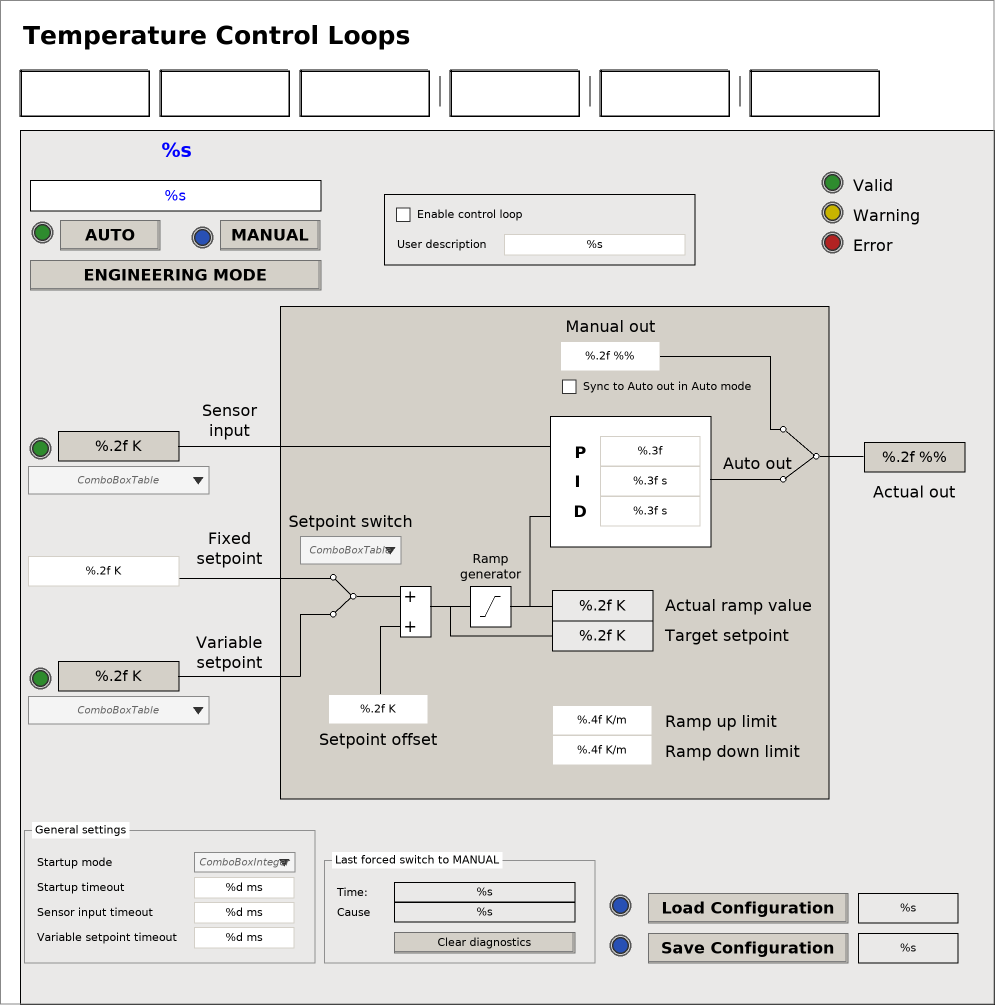
VISUALIZATION VISU_HMI_CRY_TCTRL  // 995x1005
VAR_IN_OUT
	m_Instance : FB_METIS_TCTRL;
    m_Hmi : FB_HMI_CRY_TCTRL;
    m_temp : FB_METIS_TEMPERATURES;
END_VAR
    Rectangle (20,130 975x875)
    Frame (20,70 131x48)
        shows VISU_HMI_SUBSYSTEM_BUTTON(m_Hmi := m_Hmi.tc_cry_sha_button)
        OnMouseClick: execute { m_Hmi.eActiveTab := E_HMI_CRY_TC_TABS.TC_CRY_SHA; }
    Frame (160,70 131x48)
        shows VISU_HMI_SUBSYSTEM_BUTTON(m_Hmi := m_Hmi.tc_cry_shb_button)
        OnMouseClick: execute { m_Hmi.eActiveTab := E_HMI_CRY_TC_TABS.TC_CRY_SHB; }
    Frame (300,70 131x48)
        shows VISU_HMI_SUBSYSTEM_BUTTON(m_Hmi := m_Hmi.tc_cry_shc_button)
        OnMouseClick: execute { m_Hmi.eActiveTab := E_HMI_CRY_TC_TABS.TC_CRY_SHC; }
    Frame (450,70 131x48)
        shows VISU_HMI_SUBSYSTEM_BUTTON(m_Hmi := m_Hmi.tc_cry_pt_button)
        OnMouseClick: execute { m_Hmi.eActiveTab := E_HMI_CRY_TC_TABS.TC_CRY_PT; }
    Line (440,106) (440,76)
    Line (590,106) (590,76)
    Frame (600,70 131x48)
        shows VISU_HMI_SUBSYSTEM_BUTTON(m_Hmi := m_Hmi.tc_cry_wi_button)
        OnMouseClick: execute { m_Hmi.eActiveTab := E_HMI_CRY_TC_TABS.TC_CRY_WI; }
    Frame (20,130 975x875), frame switch variable: m_Hmi.eActiveTab
        shows TEMPLATE_METIS_CTRL_TEMPERATURE(m_instance := m_Instance.tc_cry_sha, m_temp := m_temp)
        shows TEMPLATE_METIS_CTRL_TEMPERATURE(m_instance := m_Instance.tc_cry_shb, m_temp := m_temp)
        shows TEMPLATE_METIS_CTRL_TEMPERATURE(m_instance := m_Instance.tc_cry_shc, m_temp := m_temp)
        shows TEMPLATE_METIS_CTRL_TEMPERATURE(m_instance := m_Instance.tc_cry_pt, m_temp := m_temp)
        shows TEMPLATE_METIS_CTRL_TEMPERATURE(m_instance := m_Instance.tc_cry_wi, m_temp := m_temp)
        shows TEMPLATE_METIS_CTRL_TEMPERATURE(m_instance := m_Instance.tc_cry_sp, m_temp := m_temp)
    Frame (750,70 131x48)
        shows VISU_HMI_SUBSYSTEM_BUTTON(m_Hmi := m_Hmi.tc_cry_sp_button)
        OnMouseClick: execute { m_Hmi.eActiveTab := E_HMI_CRY_TC_TABS.TC_CRY_SP; }
    Line (740,106) (740,76)
    Label (20,20 411x30), "Temperature Control Loops"
END_VISUALIZATION

// HMI/VISUs/Subsystems/CRY/Components/VISU_HMI_CRY_TEMPERATURES
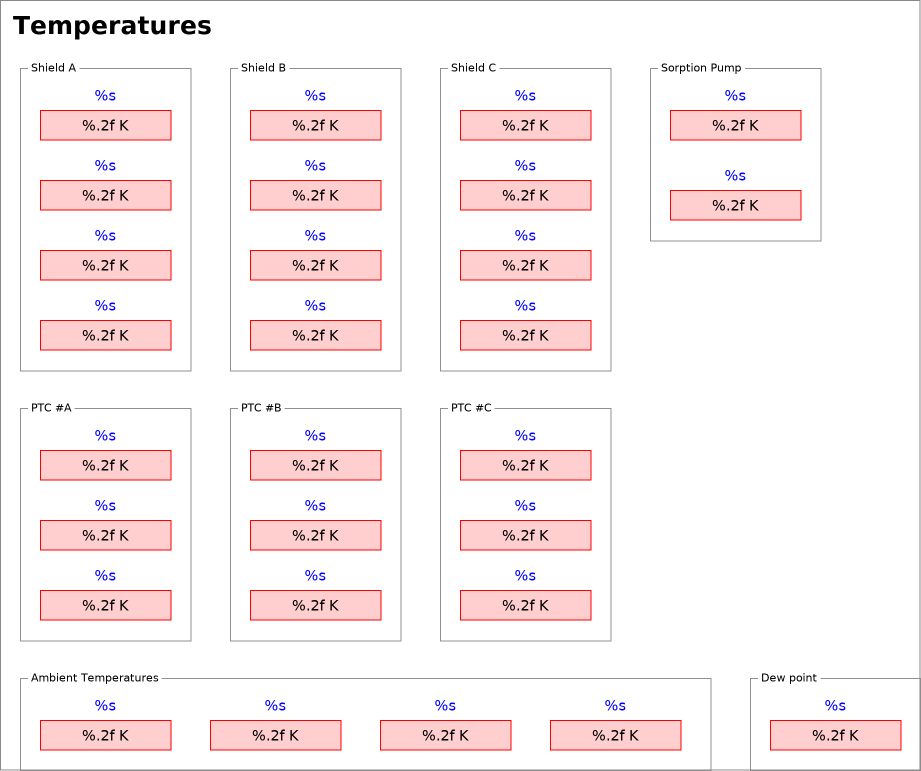
VISUALIZATION VISU_HMI_CRY_TEMPERATURES  // 921x771
VAR_IN_OUT
	m_Instance : FB_METIS_TEMPERATURES;
END_VAR
    Label (10,10 299x30), "Temperatures"
    GroupBox (20,60 171x311), "Shield A"
        Frame (10,20 150x70)
            shows TEMPLATE_TEMP_SENSOR_VALUE_ONLY(m_instance := m_Instance.t_cry_sha_1)
        Frame (10,90 150x70)
            shows TEMPLATE_TEMP_SENSOR_VALUE_ONLY(m_instance := m_Instance.t_cry_sha_2)
        Frame (10,160 150x70)
            shows TEMPLATE_TEMP_SENSOR_VALUE_ONLY(m_instance := m_Instance.t_cry_sha_3)
        Frame (10,230 150x70)
            shows TEMPLATE_TEMP_SENSOR_VALUE_ONLY(m_instance := m_Instance.t_cry_sha_4)
    GroupBox (20,400 171x241), "PTC #A"
        Frame (10,20 150x70)
            shows TEMPLATE_TEMP_SENSOR_VALUE_ONLY(m_instance := m_Instance.t_cry_pta_1)
        Frame (10,90 150x70)
            shows TEMPLATE_TEMP_SENSOR_VALUE_ONLY(m_instance := m_Instance.t_cry_pta_2)
        Frame (10,160 150x70)
            shows TEMPLATE_TEMP_SENSOR_VALUE_ONLY(m_instance := m_Instance.t_cry_pta_3)
    GroupBox (230,60 171x311), "Shield B"
        Frame (10,20 150x70)
            shows TEMPLATE_TEMP_SENSOR_VALUE_ONLY(m_instance := m_Instance.t_cry_shb_1)
        Frame (10,90 150x70)
            shows TEMPLATE_TEMP_SENSOR_VALUE_ONLY(m_instance := m_Instance.t_cry_shb_2)
        Frame (10,160 150x70)
            shows TEMPLATE_TEMP_SENSOR_VALUE_ONLY(m_instance := m_Instance.t_cry_shb_3)
        Frame (10,230 150x70)
            shows TEMPLATE_TEMP_SENSOR_VALUE_ONLY(m_instance := m_Instance.t_cry_shb_4)
    GroupBox (230,400 171x241), "PTC #B"
        Frame (10,20 150x70)
            shows TEMPLATE_TEMP_SENSOR_VALUE_ONLY(m_instance := m_Instance.t_cry_ptb_1)
        Frame (10,90 150x70)
            shows TEMPLATE_TEMP_SENSOR_VALUE_ONLY(m_instance := m_Instance.t_cry_ptb_2)
        Frame (10,160 150x70)
            shows TEMPLATE_TEMP_SENSOR_VALUE_ONLY(m_instance := m_Instance.t_cry_ptb_3)
    GroupBox (440,60 171x311), "Shield C"
        Frame (10,230 150x70)
            shows TEMPLATE_TEMP_SENSOR_VALUE_ONLY(m_instance := m_Instance.t_cry_shc_4)
        Frame (10,160 150x70)
            shows TEMPLATE_TEMP_SENSOR_VALUE_ONLY(m_instance := m_Instance.t_cry_shc_3)
        Frame (10,90 150x70)
            shows TEMPLATE_TEMP_SENSOR_VALUE_ONLY(m_instance := m_Instance.t_cry_shc_2)
        Frame (10,20 150x70)
            shows TEMPLATE_TEMP_SENSOR_VALUE_ONLY(m_instance := m_Instance.t_cry_shc_1)
    GroupBox (440,400 171x241), "PTC #C"
        Frame (10,20 150x70)
            shows TEMPLATE_TEMP_SENSOR_VALUE_ONLY(m_instance := m_Instance.t_cry_ptc_1)
        Frame (10,90 150x70)
            shows TEMPLATE_TEMP_SENSOR_VALUE_ONLY(m_instance := m_Instance.t_cry_ptc_2)
        Frame (10,160 150x70)
            shows TEMPLATE_TEMP_SENSOR_VALUE_ONLY(m_instance := m_Instance.t_cry_ptc_3)
    GroupBox (650,60 171x181), "Sorption Pump"
        Frame (10,20 150x70)
            shows TEMPLATE_TEMP_SENSOR_VALUE_ONLY(m_instance := m_Instance.t_cry_sp_1)
        Frame (10,100 150x70)
            shows TEMPLATE_TEMP_SENSOR_VALUE_ONLY(m_instance := m_Instance.t_cry_sp_2)
    GroupBox (20,670 691x101), "Ambient Temperatures"
        Frame (10,20 150x70)
            shows TEMPLATE_TEMP_SENSOR_VALUE_ONLY(m_instance := m_Instance.t_cry_pca)
        Frame (180,20 150x70)
            shows TEMPLATE_TEMP_SENSOR_VALUE_ONLY(m_instance := m_Instance.t_cry_pcb)
        Frame (350,20 150x70)
            shows TEMPLATE_TEMP_SENSOR_VALUE_ONLY(m_instance := m_Instance.t_cry_wim)
        Frame (520,20 150x70)
            shows TEMPLATE_TEMP_SENSOR_VALUE_ONLY(m_instance := m_Instance.t_cry_wia)
    GroupBox (750,670 171x101), "Dew point"
        Frame (10,20 150x70)
            shows TEMPLATE_TEMP_SENSOR_VALUE_ONLY(m_instance := m_Instance.t_cry_wid)
END_VISUALIZATION

// HMI/VISUs/Subsystems/CRY/Components/VISU_HMI_CRY_VOTERS
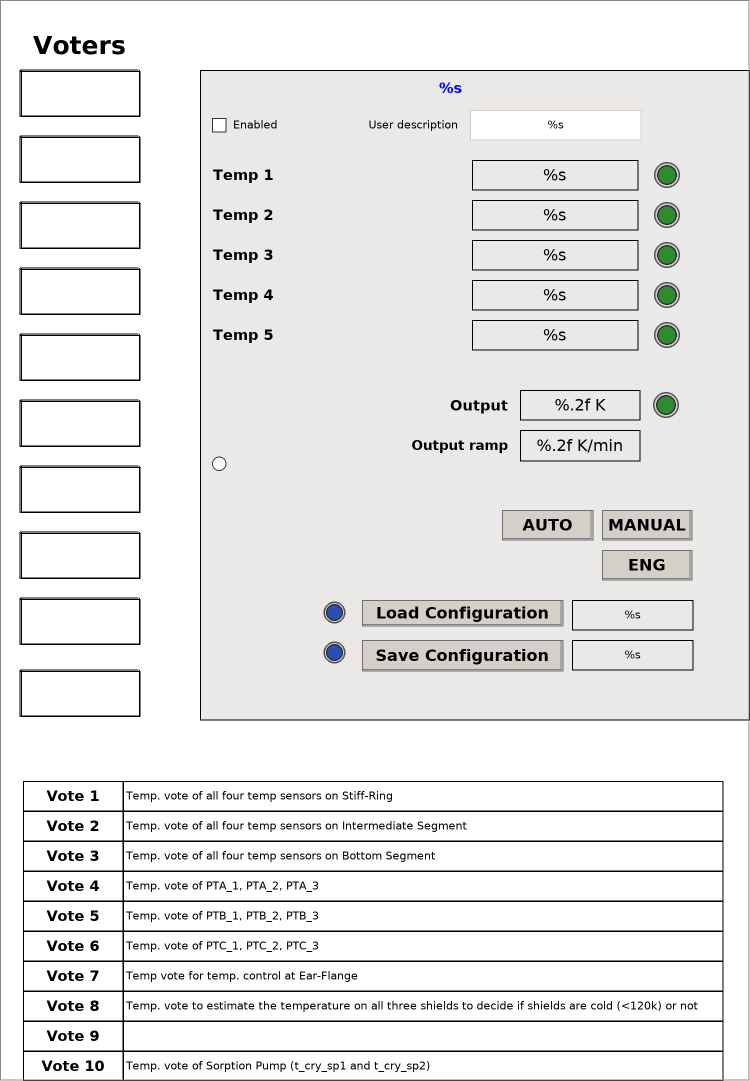
VISUALIZATION VISU_HMI_CRY_VOTERS  // 750x1081
VAR_IN_OUT
    m_Instance : FB_METIS_VOTERS;
	m_Hmi : FB_HMI_CRY_VOTERS;
    m_temperatures : FB_METIS_TEMPERATURES;
END_VAR
    Rectangle (200,70 550x650)
    Frame (20,70 121x48)
        shows VISU_HMI_SUBSYSTEM_BUTTON(m_Hmi := m_Hmi.fbVoter1Button)
        OnMouseClick: execute { m_Hmi.eActiveTab := E_HMI_VOTER_TABS.VOTER_1; }
    Frame (20,136 121x48)
        shows VISU_HMI_SUBSYSTEM_BUTTON(m_Hmi := m_Hmi.fbVoter2Button)
        OnMouseClick: execute { m_Hmi.eActiveTab := E_HMI_VOTER_TABS.VOTER_2; }
    Frame (20,202 121x48)
        shows VISU_HMI_SUBSYSTEM_BUTTON(m_Hmi := m_Hmi.fbVoter3Button)
        OnMouseClick: execute { m_Hmi.eActiveTab := E_HMI_VOTER_TABS.VOTER_3; }
    Frame (20,268 121x48)
        shows VISU_HMI_SUBSYSTEM_BUTTON(m_Hmi := m_Hmi.fbVoter4Button)
        OnMouseClick: execute { m_Hmi.eActiveTab := E_HMI_VOTER_TABS.VOTER_4; }
    Frame (20,334 121x48)
        shows VISU_HMI_SUBSYSTEM_BUTTON(m_Hmi := m_Hmi.fbVoter5Button)
        OnMouseClick: execute { m_Hmi.eActiveTab := E_HMI_VOTER_TABS.VOTER_5; }
    Frame (20,400 121x48)
        shows VISU_HMI_SUBSYSTEM_BUTTON(m_Hmi := m_Hmi.fbVoter6Button)
        OnMouseClick: execute { m_Hmi.eActiveTab := E_HMI_VOTER_TABS.VOTER_6; }
    Frame (20,466 121x48)
        shows VISU_HMI_SUBSYSTEM_BUTTON(m_Hmi := m_Hmi.fbVoter7Button)
        OnMouseClick: execute { m_Hmi.eActiveTab := E_HMI_VOTER_TABS.VOTER_7; }
    Frame (20,532 121x48)
        shows VISU_HMI_SUBSYSTEM_BUTTON(m_Hmi := m_Hmi.fbVoter8Button)
        OnMouseClick: execute { m_Hmi.eActiveTab := E_HMI_VOTER_TABS.VOTER_8; }
    Frame (20,598 121x48)
        shows VISU_HMI_SUBSYSTEM_BUTTON(m_Hmi := m_Hmi.fbVoter9Button)
        OnMouseClick: execute { m_Hmi.eActiveTab := E_HMI_VOTER_TABS.VOTER_9; }
    Frame (20,670 121x48)
        shows VISU_HMI_SUBSYSTEM_BUTTON(m_Hmi := m_Hmi.fbVoter10Button)
        OnMouseClick: execute { m_Hmi.eActiveTab := E_HMI_VOTER_TABS.VOTER_10; }
    Frame (200,70 545x641), frame switch variable: m_Hmi.eActiveTab
        shows TEMPLATE_TEMPERATURE_VOTE(m_Instance := m_Instance.vote_cry_1, m_all_temperatures_array := m_temperatures)
        shows TEMPLATE_TEMPERATURE_VOTE(m_Instance := m_Instance.vote_cry_2, m_all_temperatures_array := m_temperatures)
        shows TEMPLATE_TEMPERATURE_VOTE(m_Instance := m_Instance.vote_cry_3, m_all_temperatures_array := m_temperatures)
        shows TEMPLATE_TEMPERATURE_VOTE(m_Instance := m_Instance.vote_cry_4, m_all_temperatures_array := m_temperatures)
        shows TEMPLATE_TEMPERATURE_VOTE(m_Instance := m_Instance.vote_cry_5, m_all_temperatures_array := m_temperatures)
        shows TEMPLATE_TEMPERATURE_VOTE(m_Instance := m_Instance.vote_cry_6, m_all_temperatures_array := m_temperatures)
        shows TEMPLATE_TEMPERATURE_VOTE(m_Instance := m_Instance.vote_cry_7, m_all_temperatures_array := m_temperatures)
        shows TEMPLATE_TEMPERATURE_VOTE(m_Instance := m_Instance.vote_cry_8, m_all_temperatures_array := m_temperatures)
        shows TEMPLATE_TEMPERATURE_VOTE(m_Instance := m_Instance.vote_cry_9, m_all_temperatures_array := m_temperatures)
        shows TEMPLATE_TEMPERATURE_VOTE(m_Instance := m_Instance.vote_cry_10, m_all_temperatures_array := m_temperatures)
    Label (30,30 411x30), "Voters"
    Rectangle (23,781 100x30), "Vote 1"
    Rectangle (123,781 600x30), "Temp. vote of all four temp sensors on Stiff-Ring"
    Rectangle (23,811 100x30), "Vote 2"
    Rectangle (123,811 600x30), "Temp. vote of all four temp sensors on Intermediate Segment"
    Rectangle (23,841 100x30), "Vote 3"
    Rectangle (123,841 600x30), "Temp. vote of all four temp sensors on Bottom Segment"
    Rectangle (23,871 100x30), "Vote 4"
    Rectangle (123,871 600x30), "Temp. vote of PTA_1, PTA_2, PTA_3"
    Rectangle (23,901 100x30), "Vote 5"
    Rectangle (123,901 600x30), "Temp. vote of PTB_1, PTB_2, PTB_3"
    Rectangle (23,931 100x30), "Vote 6"
    Rectangle (123,931 600x30), "Temp. vote of PTC_1, PTC_2, PTC_3"
    Rectangle (23,961 100x30), "Vote 7"
    Rectangle (123,961 600x30), "Temp vote for temp. control at Ear-Flange"
    Rectangle (23,991 100x30), "Vote 8"
    Rectangle (123,991 600x30), "Temp. vote to estimate the temperature on all three shields to decide if shields are cold (<120k) or not"
    Rectangle (23,1021 100x30), "Vote 9"
    Rectangle (123,1021 600x30)
    Rectangle (23,1051 100x30), "Vote 10"
    Rectangle (123,1051 600x30), "Temp. vote of Sorption Pump (t_cry_sp1 and t_cry_sp2)"
END_VISUALIZATION

// HMI/VISUs/Subsystems/CRY/VISU_HMI_CRY
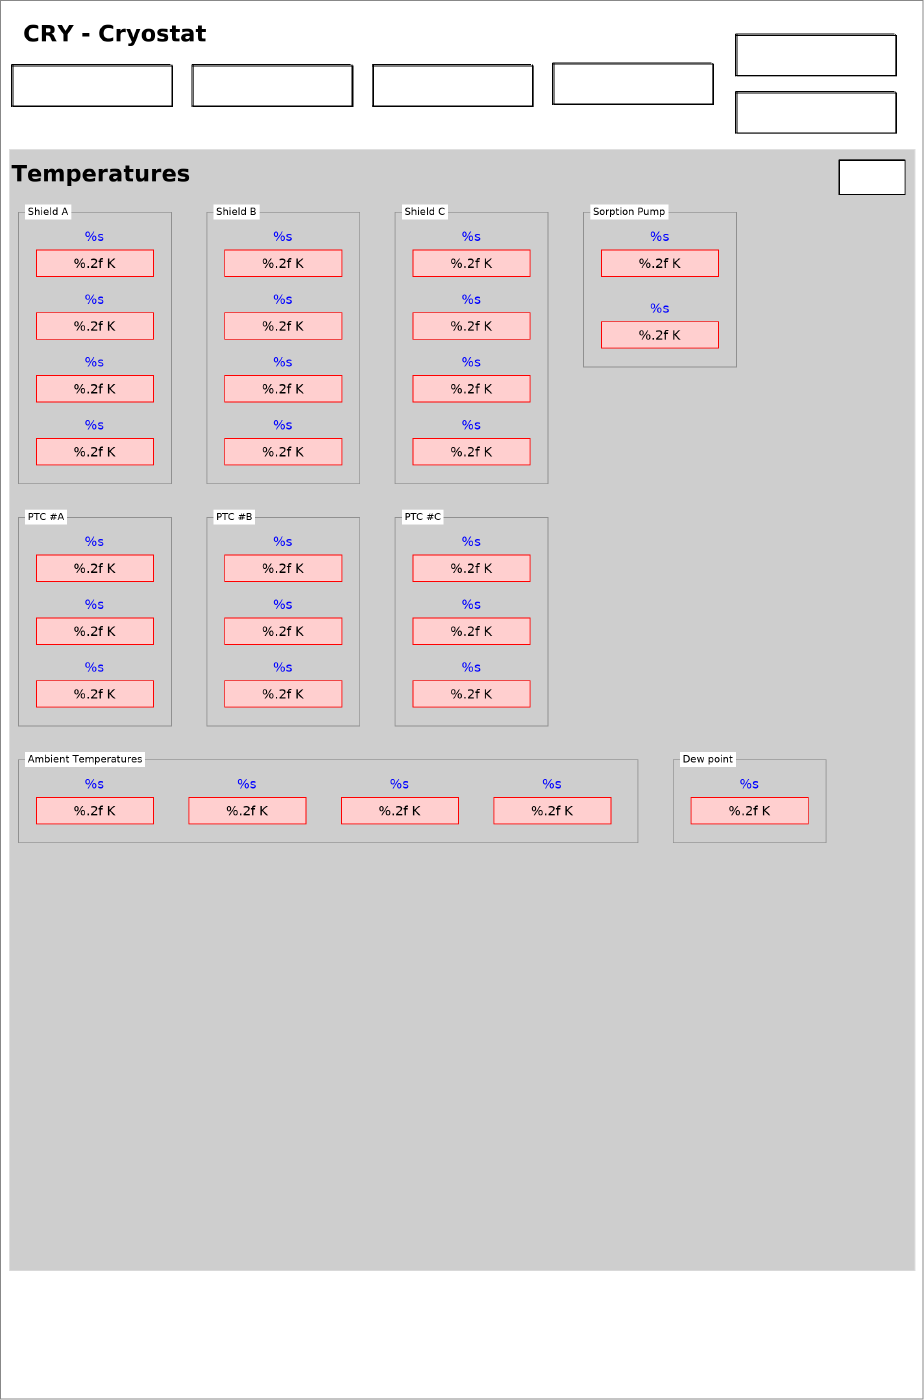
VISUALIZATION VISU_HMI_CRY  // 1030x1560
VAR_IN_OUT
	met_cryo_ctrl: FB_METIS_CRYO_CTRL;
    m_Hmi : FB_HMI_CRY;
END_VAR
    Frame (0,36 1021x1397)
        shows TEMPLATE_BACKGROUND_LEVEL_2()
    Label (23,22 671x30), "CRY - Cryostat"
    Frame (0,168 1017x1250), frame switch variable: m_Hmi.eActiveTab
        shows VISU_HMI_CRY_TEMPERATURES(m_Instance := met_cryo_ctrl.met_temp)
        shows VISU_HMI_CRY_RH(m_Instance := met_cryo_ctrl.met_rh)
        shows VISU_HMI_CRY_HEATERS(m_Instance := met_cryo_ctrl.met_heaters, m_Hmi := m_Hmi.fbHeaters)
        shows VISU_HMI_CRY_VOTERS(m_Instance := met_cryo_ctrl.met_voters, m_Hmi := m_Hmi.fbVoters, m_temperatures := met_cryo_ctrl.met_temp)
        shows VISU_HMI_CRY_TCTRL(m_Instance := met_cryo_ctrl.met_tctrl, m_Hmi := m_Hmi.fbTControl, m_temp := met_cryo_ctrl.met_temp)
        shows VISU_HMI_CRY_LN2_LEVEL_CONTROL()
    Frame (13,72 181x48)
        shows VISU_HMI_SUBSYSTEM_BUTTON(m_Hmi := m_Hmi.fbTemperaturesButton)
        OnMouseClick: execute { m_Hmi.eActiveTab := E_HMI_CRY_TABS.TEMPERATURES; }
    Frame (616,70 181x48)
        shows VISU_HMI_SUBSYSTEM_BUTTON(m_Hmi := m_Hmi.fbHeatersButton)
        OnMouseClick: execute { m_Hmi.eActiveTab := E_HMI_CRY_TABS.HEATERS; }
    Frame (214,72 181x48)
        shows VISU_HMI_SUBSYSTEM_BUTTON(m_Hmi := m_Hmi.fbVotersButton)
        OnMouseClick: execute { m_Hmi.eActiveTab := E_HMI_CRY_TABS.VOTERS; }
    Frame (415,72 181x48)
        shows VISU_HMI_SUBSYSTEM_BUTTON(m_Hmi := m_Hmi.fbTControlButton)
        OnMouseClick: execute { m_Hmi.eActiveTab := E_HMI_CRY_TABS.TCONTROL; }
    Group (820,38 181x112)
        Frame (0,0 181x48)
            shows VISU_HMI_SUBSYSTEM_BUTTON(m_Hmi := m_Hmi.fbRhButton)
            OnMouseClick: execute { m_Hmi.eActiveTab := E_HMI_CRY_TABS.RH; }
        Frame (0,64 181x48)
            shows VISU_HMI_SUBSYSTEM_BUTTON(m_Hmi := m_Hmi.fbLN2ControlButton)
            OnMouseClick: execute { m_Hmi.eActiveTab := E_HMI_CRY_TABS.LN2CONTROL; }
    Frame (935,178 75x40)
        shows VISU_HMI_SUBSYSTEM_BUTTON(m_Hmi := PRG_HMI.fbBackButton)
        OnMouseClick: execute { PRG_HMI.eActiveTab := PRG_HMI.ePreviousTab; }
END_VISUALIZATION

// HMI/VISUs/Subsystems/ICS/Components/VISU_HMI_ICS_CCU_CONFIGS
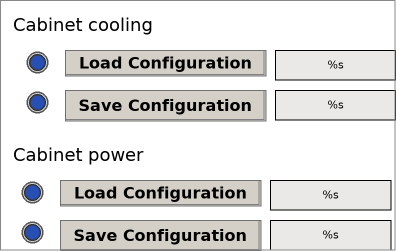
VISUALIZATION VISU_HMI_ICS_CCU_CONFIGS  // 396x251
VAR_IN_OUT
	m_CoolingCfg : FB_READ_WRITE_CAB_COOLING_CONFIG;
    m_PowerCfg : FB_READ_WRITE_CAB_POWER_CONFIG;
END_VAR
    Lamp1 (25,50 25x25), tooltip "Command coming from the Control System", variable: m_CoolingCfg.bReading, style: Lamp-Lamp1-Blue
    Button (65,90 201x31), "Save Configuration"
        OnMouseClick: execute { m_CoolingCfg.M_WriteConfiguration(); }
    Button (65,50 201x26), "Load Configuration"
        OnMouseClick: execute { m_CoolingCfg.M_ReadConfiguration(); }
    Lamp1 (25,90 25x25), tooltip "Command coming from the Control System", variable: m_CoolingCfg.bWriting, style: Lamp-Lamp1-Blue
    Rectangle (275,50 121x30), "%s", text variable: m_CoolingCfg.sReadError, colour toggle: m_CoolingCfg.bReadError
    Rectangle (275,90 121x30), "%s", text variable: m_CoolingCfg.sWriteError, colour toggle: m_CoolingCfg.bWriteError
    Label (10,10 206x30), "Cabinet cooling"
    Label (10,140 206x30), "Cabinet power"
    Lamp1 (20,180 25x25), variable: m_PowerCfg.bReading, style: Lamp-Lamp1-Blue
    Button (60,220 201x31), "Save Configuration"
        OnMouseClick: execute { m_PowerCfg.M_WriteConfiguration(); }
    Button (60,180 201x26), "Load Configuration"
        OnMouseClick: execute { m_PowerCfg.M_ReadConfiguration(); }
    Lamp1 (20,220 25x25), tooltip "Command coming from the Control System", variable: m_PowerCfg.bWriting, style: Lamp-Lamp1-Blue
    Rectangle (270,180 121x30), "%s", text variable: m_PowerCfg.sReadError, colour toggle: m_PowerCfg.bReadError
    Rectangle (270,220 121x30), "%s", text variable: m_PowerCfg.sWriteError, colour toggle: m_PowerCfg.bWriteError
END_VISUALIZATION

// HMI/VISUs/Subsystems/ICS/Components/VISU_HMI_ICS_CCUS_CONFIGS
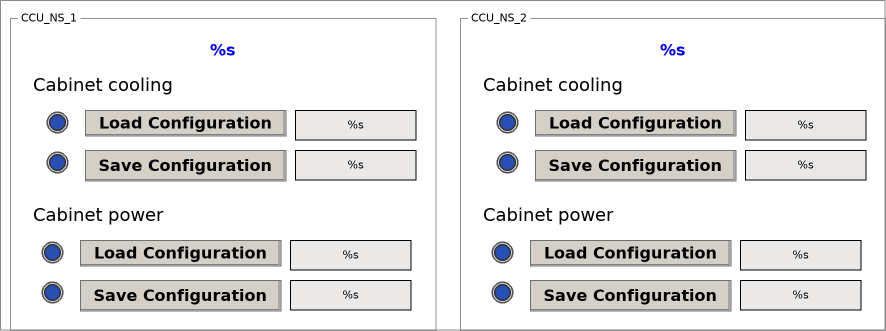
VISUALIZATION VISU_HMI_ICS_CCUS_CONFIGS  // 886x331
VAR_IN_OUT
	m_CCUs : FB_METIS_CCUS;
    m_Hmi : FB_HMI_ICS;
END_VAR
    GroupBox (10,10 426x321), "CCU_NS_1"
        Frame (10,50 397x252)
            shows VISU_HMI_ICS_CCU_CONFIGS(m_CoolingCfg := m_CCUs.aCoolingConfig[1], m_PowerCfg := m_CCUs.aPowerConfig[1])
        Rectangle (20,25 386x30), "%s", text variable: m_CCUs.ccu_ns_1.in_sCabinetName
    GroupBox (460,10 426x321), "CCU_NS_2"
        Frame (10,50 397x252)
            shows VISU_HMI_ICS_CCU_CONFIGS(m_CoolingCfg := m_CCUs.aCoolingConfig[2], m_PowerCfg := m_CCUs.aPowerConfig[2])
        Rectangle (20,25 386x30), "%s", text variable: m_CCUs.ccu_ns_2.in_sCabinetName
END_VISUALIZATION

// HMI/VISUs/Subsystems/ICS/VISU_HMI_ICS
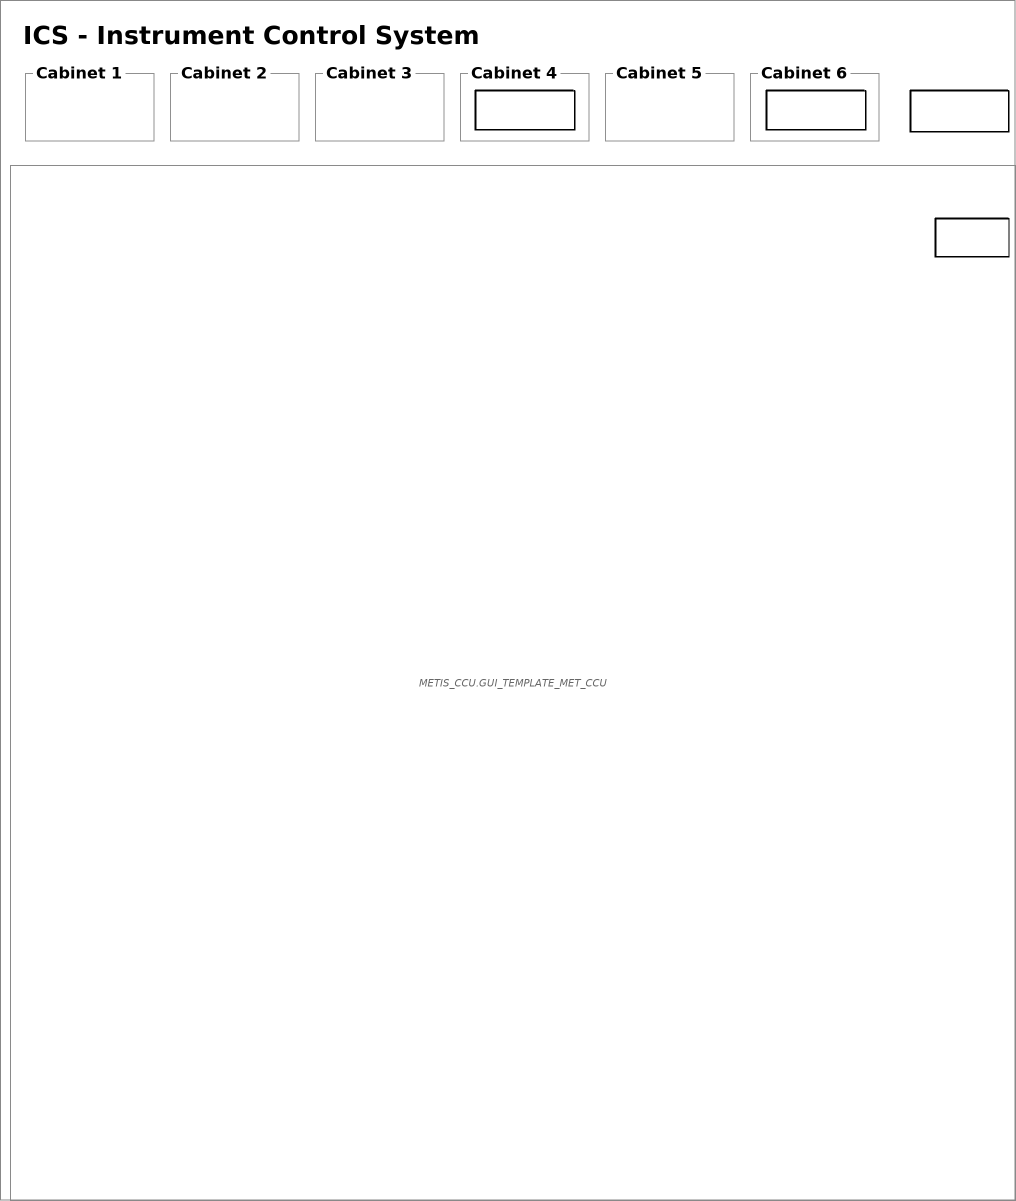
VISUALIZATION VISU_HMI_ICS  // 1016x1201
VAR_IN_OUT
	m_CCUs : FB_METIS_CCUS;
    m_Hmi : FB_HMI_ICS;
END_VAR
    Label (20,20 671x30), "ICS - Instrument Control System"
    Frame (10,165 1006x1036), frame switch variable: m_Hmi.eActiveTab
        shows METIS_CCU.GUI_TEMPLATE_MET_CCU(m_Instance := m_CCUs.ccu_ns_1)
        shows METIS_CCU.GUI_TEMPLATE_MET_CCU(m_Instance := m_CCUs.ccu_ns_2)
        shows VISU_HMI_ICS_CCUS_CONFIGS(m_CCUs := m_CCUs, m_Hmi := m_Hmi)
        shows METIS_CCU.GUI_TEMPLATE_MET_CCU(m_Instance := m_CCUs.ccu_ns_4)
        shows METIS_CCU.GUI_TEMPLATE_MET_CCU(m_Instance := m_CCUs.ccu_ns_5)
        shows METIS_CCU.GUI_TEMPLATE_MET_CCU(m_Instance := m_CCUs.ccu_6)
        shows VISU_HMI_ICS_CCUS_CONFIGS(m_CCUs := m_CCUs, m_Hmi := m_Hmi)
        p4089929901: m_CCUs.ccu_ns_3
    Frame (910,90 100x43)
        shows VISU_HMI_SUBSYSTEM_BUTTON(m_Hmi := m_Hmi.fbConfigsButton)
        shows METIS_CCU.GUI_TEMPLATE_MET_CCU()
        shows METIS_CCU.GUI_TEMPLATE_MET_CCU()
        shows METIS_CCU.GUI_TEMPLATE_MET_CCU()
        shows METIS_CCU.GUI_TEMPLATE_MET_CCU()
        shows METIS_CCU.GUI_TEMPLATE_MET_CCU()
        OnMouseClick: execute { m_Hmi.eActiveTab := E_HMI_ICS_TABS.CCU_CONFIGS; }
    Frame (935,218 75x40)
        shows VISU_HMI_SUBSYSTEM_BUTTON(m_Hmi := PRG_HMI.fbBackButton)
        OnMouseClick: execute { PRG_HMI.eActiveTab := PRG_HMI.ePreviousTab; }
    GroupBox (25,65 129x76), "Cabinet 1"
    GroupBox (170,65 129x76), "Cabinet 2"
    GroupBox (315,65 129x76), "Cabinet 3"
    GroupBox (460,65 129x76), "Cabinet 4"
        Frame (15,25 101x41)
            shows VISU_HMI_SUBSYSTEM_BUTTON(m_Hmi := m_Hmi.fbCCU_NS_2_Button)
            shows METIS_CCU.GUI_TEMPLATE_MET_CCU()
            shows METIS_CCU.GUI_TEMPLATE_MET_CCU()
            shows METIS_CCU.GUI_TEMPLATE_MET_CCU()
            shows METIS_CCU.GUI_TEMPLATE_MET_CCU()
            shows METIS_CCU.GUI_TEMPLATE_MET_CCU()
            OnMouseClick: execute { m_Hmi.eActiveTab := E_HMI_ICS_TABS.CCU_NS_2; }
    GroupBox (605,65 129x76), "Cabinet 5"
    GroupBox (750,65 129x76), "Cabinet 6"
        Frame (16,25 101x41)
            shows VISU_HMI_SUBSYSTEM_BUTTON(m_Hmi := m_Hmi.fbCCU_NS_1_Button)
            shows METIS_CCU.GUI_TEMPLATE_MET_CCU()
            shows METIS_CCU.GUI_TEMPLATE_MET_CCU()
            shows METIS_CCU.GUI_TEMPLATE_MET_CCU()
            shows METIS_CCU.GUI_TEMPLATE_MET_CCU()
            shows METIS_CCU.GUI_TEMPLATE_MET_CCU()
            OnMouseClick: execute { m_Hmi.eActiveTab := E_HMI_ICS_TABS.CCU_NS_1; }
END_VISUALIZATION

// HMI/VISUs/Subsystems/IMG/Components/VISU_HMI_IMG_HEATERS
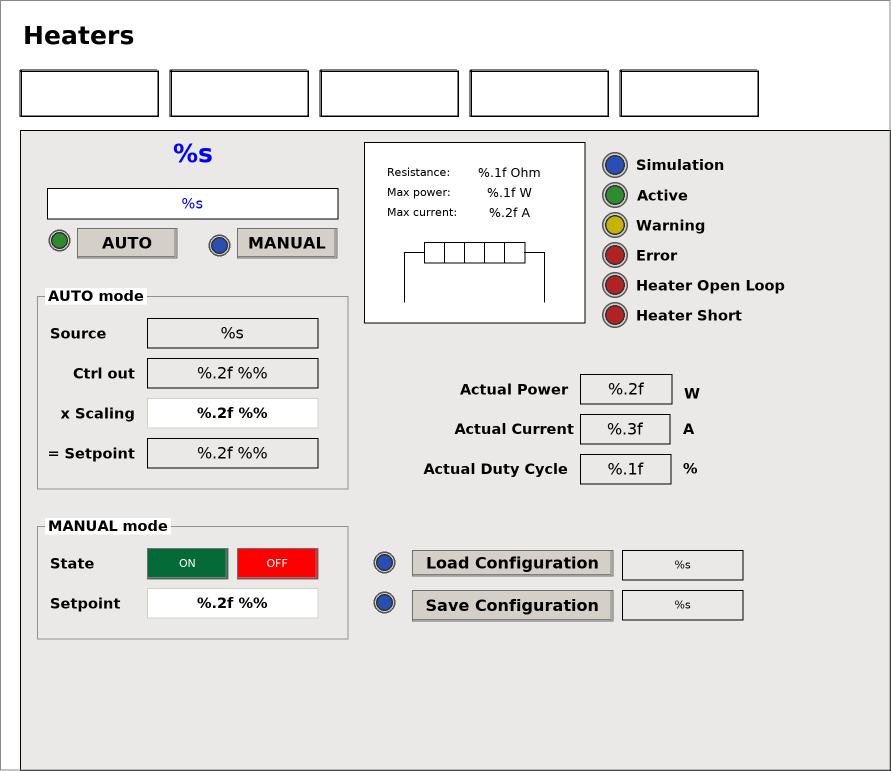
VISUALIZATION VISU_HMI_IMG_HEATERS  // 891x771
VAR_IN_OUT
	m_Instance  : FB_METIS_HEATERS;
    m_Hmi       : FB_HMI_IMG_HEATERS;
END_VAR
    Rectangle (20,130 871x641)
    Label (20,20 411x30), "Heaters"
    Frame (20,130 800x550), frame switch variable: m_Hmi.eActiveTab
        shows TEMPLATE_METIS_HEATER(m_instance := m_Instance.h_img_wuh_1)
        shows TEMPLATE_METIS_HEATER(m_instance := m_Instance.h_img_wuh_2)
        shows TEMPLATE_METIS_HEATER(m_instance := m_Instance.h_img_lmd_2)
        shows TEMPLATE_METIS_HEATER(m_instance := m_Instance.h_img_lmp_2)
        shows TEMPLATE_METIS_HEATER(m_instance := m_Instance.h_img_nd_2)
        shows METIS_Cryo_PLC.TEMPLATE_METIS_CTRL_DT670(m_temp := m_temp)
        p8630679: tcontrol.tc_img_wuh_1
        p371692913: tcontrol.vote_img_wuh_1
        p2286783886: temperatures
    Frame (20,70 140x48)
        shows VISU_HMI_SUBSYSTEM_BUTTON(m_Hmi := m_Hmi.h_img_wuh_1_button)
        OnMouseClick: execute { m_Hmi.eActiveTab := E_HMI_IMG_HEATER_TABS.H_IMG_WUH_1; }
    Frame (170,70 140x48)
        shows VISU_HMI_SUBSYSTEM_BUTTON(m_Hmi := m_Hmi.h_img_wuh_2_button)
        OnMouseClick: execute { m_Hmi.eActiveTab := E_HMI_IMG_HEATER_TABS.H_IMG_WUH_2; }
    Frame (320,70 140x48)
        shows VISU_HMI_SUBSYSTEM_BUTTON(m_Hmi := m_Hmi.h_img_lmd_2_button)
        OnMouseClick: execute { m_Hmi.eActiveTab := E_HMI_IMG_HEATER_TABS.H_IMG_LMD_2; }
    Frame (470,70 140x48)
        shows VISU_HMI_SUBSYSTEM_BUTTON(m_Hmi := m_Hmi.h_img_lmp_2_button)
        OnMouseClick: execute { m_Hmi.eActiveTab := E_HMI_IMG_HEATER_TABS.H_IMG_LMP_2; }
    Frame (620,70 140x48)
        shows VISU_HMI_SUBSYSTEM_BUTTON(m_Hmi := m_Hmi.h_img_nd_2_button)
        OnMouseClick: execute { m_Hmi.eActiveTab := E_HMI_IMG_HEATER_TABS.H_IMG_ND_2; }
END_VISUALIZATION

// HMI/VISUs/Subsystems/IMG/Components/VISU_HMI_IMG_TC
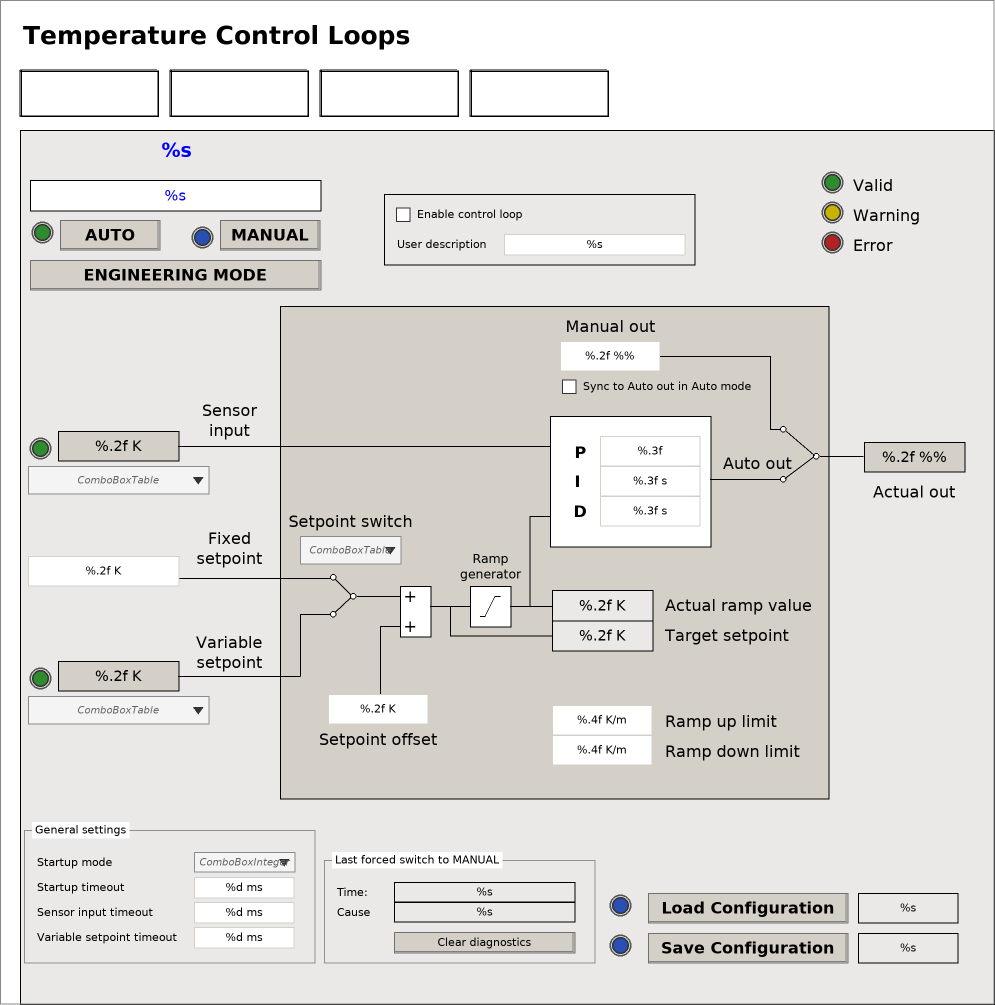
VISUALIZATION VISU_HMI_IMG_TC  // 995x1005
VAR_IN_OUT
    m_Instance : FB_METIS_TCTRL;
    m_Hmi : FB_HMI_IMG_TCTRL;
    m_temp : FB_METIS_TEMPERATURES;
END_VAR
    Rectangle (20,130 975x875)
    Label (20,20 411x30), "Temperature Control Loops"
    Frame (20,130 975x875), frame switch variable: m_Hmi.eActiveTab
        shows TEMPLATE_METIS_CTRL_TEMPERATURE(m_instance := m_Instance.tc_img_wuh, m_temp := m_temp)
        shows TEMPLATE_METIS_CTRL_TEMPERATURE(m_instance := m_Instance.tc_img_lmd_2, m_temp := m_temp)
        shows TEMPLATE_METIS_CTRL_TEMPERATURE(m_instance := m_Instance.tc_img_lmp_2, m_temp := m_temp)
        shows TEMPLATE_METIS_CTRL_TEMPERATURE(m_instance := m_Instance.tc_img_nd_2, m_temp := m_temp)
        shows METIS_Cryo_PLC.TEMPLATE_METIS_CTRL_DT670(m_temp := m_temp)
        p8630679: tcontrol.tc_img_wuh_1
        p371692913: tcontrol.vote_img_wuh_1
        p2286783886: temperatures
        p2857688358: m_Instance.tc_img_nd_2
        p3792852128: m_temp
    Frame (20,70 140x48)
        shows VISU_HMI_SUBSYSTEM_BUTTON(m_Hmi := m_Hmi.tc_img_wuh_button)
        OnMouseClick: execute { m_Hmi.eActiveTab := E_HMI_IMG_TC_TABS.TC_IMG_WUH; }
    Frame (170,70 140x48)
        shows VISU_HMI_SUBSYSTEM_BUTTON(m_Hmi := m_Hmi.tc_img_lmd_2_button)
        OnMouseClick: execute { m_Hmi.eActiveTab := E_HMI_IMG_TC_TABS.TC_IMG_LMD_2; }
    Frame (320,70 140x48)
        shows VISU_HMI_SUBSYSTEM_BUTTON(m_Hmi := m_Hmi.tc_img_lmp_2_button)
        OnMouseClick: execute { m_Hmi.eActiveTab := E_HMI_IMG_TC_TABS.TC_IMG_LMP_2; }
    Frame (470,70 140x48)
        shows VISU_HMI_SUBSYSTEM_BUTTON(m_Hmi := m_Hmi.tc_img_nd_2_button)
        OnMouseClick: execute { m_Hmi.eActiveTab := E_HMI_IMG_TC_TABS.TC_IMG_ND_2; }
END_VISUALIZATION

// HMI/VISUs/Subsystems/IMG/Components/VISU_HMI_IMG_TEMPERATURES
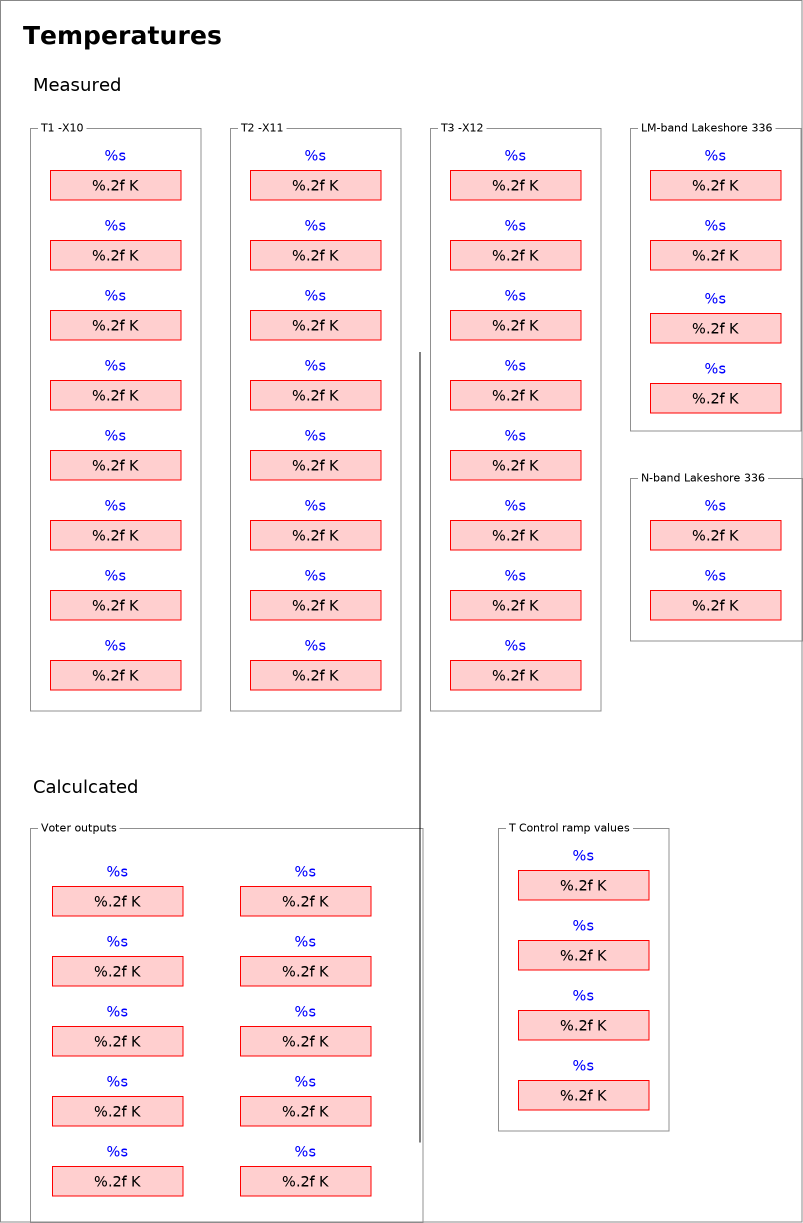
VISUALIZATION VISU_HMI_IMG_TEMPERATURES  // 803x1223
VAR_IN_OUT
	m_Instance : FB_METIS_TEMPERATURES;
END_VAR
    GroupBox (230,120 171x591), "T2 -X11"
        Frame (10,20 150x70)
            shows TEMPLATE_TEMP_SENSOR_VALUE_ONLY(m_instance := m_Instance.t_img_npw_1)
        Frame (10,90 150x70)
            shows TEMPLATE_TEMP_SENSOR_VALUE_ONLY(m_instance := m_Instance.t_img_npw_2)
        Frame (10,160 150x70)
            shows TEMPLATE_TEMP_SENSOR_VALUE_ONLY(m_instance := m_Instance.t_img_nfw_1)
        Frame (10,230 150x70)
            shows TEMPLATE_TEMP_SENSOR_VALUE_ONLY(m_instance := m_Instance.t_img_nfw_2)
        Frame (10,300 150x70)
            shows TEMPLATE_TEMP_SENSOR_VALUE_ONLY(m_instance := m_Instance.t_img_npr_1)
        Frame (10,370 150x70)
            shows TEMPLATE_TEMP_SENSOR_VALUE_ONLY(m_instance := m_Instance.t_img_bwu_2)
        Frame (10,440 150x70)
            shows TEMPLATE_TEMP_SENSOR_VALUE_ONLY(m_instance := m_Instance.t_img_nnd_1)
        Frame (10,510 150x70)
            shows TEMPLATE_TEMP_SENSOR_VALUE_ONLY(m_instance := m_Instance.t_img_nnd_2)
    GroupBox (30,120 171x591), "T1 -X10"
        Frame (10,20 150x70)
            shows TEMPLATE_TEMP_SENSOR_VALUE_ONLY(m_instance := m_Instance.t_img_lpw_1)
        Frame (10,90 150x70)
            shows TEMPLATE_TEMP_SENSOR_VALUE_ONLY(m_instance := m_Instance.t_img_lpw_2)
        Frame (10,160 150x70)
            shows TEMPLATE_TEMP_SENSOR_VALUE_ONLY(m_instance := m_Instance.t_img_lfw_1)
        Frame (10,230 150x70)
            shows TEMPLATE_TEMP_SENSOR_VALUE_ONLY(m_instance := m_Instance.t_img_lfw_2)
        Frame (10,300 150x70)
            shows TEMPLATE_TEMP_SENSOR_VALUE_ONLY(m_instance := m_Instance.t_img_lpr_1)
        Frame (10,370 150x70)
            shows TEMPLATE_TEMP_SENSOR_VALUE_ONLY(m_instance := m_Instance.t_img_bwu_3)
        Frame (10,440 150x70)
            shows TEMPLATE_TEMP_SENSOR_VALUE_ONLY(m_instance := m_Instance.t_img_lnd_1)
        Frame (10,510 150x70)
            shows TEMPLATE_TEMP_SENSOR_VALUE_ONLY(m_instance := m_Instance.t_img_lnd_2)
    Label (20,20 299x30), "Temperatures"
    GroupBox (430,120 171x591), "T3 -X12"
        Frame (10,20 150x70)
            shows TEMPLATE_TEMP_SENSOR_VALUE_ONLY(m_instance := m_Instance.t_img_opt_1)
        Frame (10,90 150x70)
            shows TEMPLATE_TEMP_SENSOR_VALUE_ONLY(m_instance := m_Instance.t_img_bwu_1)
        Frame (10,160 150x70)
            shows TEMPLATE_TEMP_SENSOR_VALUE_ONLY(m_instance := m_Instance.t_img_ctr_1)
        Frame (10,230 150x70)
            shows TEMPLATE_TEMP_SENSOR_VALUE_ONLY(m_instance := m_Instance.t_img_ctr_2)
        Frame (10,300 150x70)
            shows TEMPLATE_TEMP_SENSOR_VALUE_ONLY(m_instance := m_Instance.t_img_70k_1)
        Frame (10,370 150x70)
            shows TEMPLATE_TEMP_SENSOR_VALUE_ONLY(m_instance := m_Instance.t_img_ln2_1)
        Frame (10,440 150x70)
            shows TEMPLATE_TEMP_SENSOR_VALUE_ONLY(m_instance := m_Instance.t_img_ln2_2)
        Frame (10,510 150x70)
            shows TEMPLATE_TEMP_SENSOR_VALUE_ONLY(m_instance := m_Instance.t_img_hex_1)
    GroupBox (630,120 171x311), "LM-band Lakeshore 336"
        Frame (10,20 150x70)
            shows TEMPLATE_TEMP_SENSOR_VALUE_ONLY(m_instance := m_Instance.t_img_lmd_1)
        Frame (10,90 150x70)
            shows TEMPLATE_TEMP_SENSOR_VALUE_ONLY(m_instance := m_Instance.t_img_lmd_2)
        Frame (10,163 150x70)
            shows TEMPLATE_TEMP_SENSOR_VALUE_ONLY(m_instance := m_Instance.t_img_lmp_1)
        Frame (10,233 150x70)
            shows TEMPLATE_TEMP_SENSOR_VALUE_ONLY(m_instance := m_Instance.t_img_lmp_2)
    GroupBox (630,470 173x171), "N-band Lakeshore 336"
        Frame (10,20 150x70)
            shows TEMPLATE_TEMP_SENSOR_VALUE_ONLY(m_instance := m_Instance.t_img_nd_1)
        Frame (10,90 150x70)
            shows TEMPLATE_TEMP_SENSOR_VALUE_ONLY(m_instance := m_Instance.t_img_nd_2)
    GroupBox (30,820 393x403), "Voter outputs"
        Group (12,36 150x350)
            Frame (0,0 150x70)
                shows TEMPLATE_TEMP_SENSOR_VALUE_ONLY(m_instance := m_Instance.t_img_vot_1)
            Frame (0,70 150x70)
                shows TEMPLATE_TEMP_SENSOR_VALUE_ONLY(m_instance := m_Instance.t_img_vot_2)
            Frame (0,140 150x70)
                shows TEMPLATE_TEMP_SENSOR_VALUE_ONLY(m_instance := m_Instance.t_img_vot_3)
            Frame (0,210 150x70)
                shows TEMPLATE_TEMP_SENSOR_VALUE_ONLY(m_instance := m_Instance.t_img_vot_4)
            Frame (0,280 150x70)
                shows TEMPLATE_TEMP_SENSOR_VALUE_ONLY(m_instance := m_Instance.t_img_vot_5)
        Group (200,36 150x350)
            Frame (0,0 150x70)
                shows TEMPLATE_TEMP_SENSOR_VALUE_ONLY(m_instance := m_Instance.t_img_vot_6)
            Frame (0,70 150x70)
                shows TEMPLATE_TEMP_SENSOR_VALUE_ONLY(m_instance := m_Instance.t_img_vot_7)
            Frame (0,140 150x70)
                shows TEMPLATE_TEMP_SENSOR_VALUE_ONLY(m_instance := m_Instance.t_img_vot_8)
            Frame (0,210 150x70)
                shows TEMPLATE_TEMP_SENSOR_VALUE_ONLY(m_instance := m_Instance.t_img_vot_9)
            Frame (0,280 150x70)
                shows TEMPLATE_TEMP_SENSOR_VALUE_ONLY(m_instance := m_Instance.t_img_vot_10)
    GroupBox (498,820 171x311), "T Control ramp values"
        Frame (10,20 150x70)
            shows TEMPLATE_TEMP_SENSOR_VALUE_ONLY(m_instance := m_Instance.t_img_wuh_ramp)
        Frame (10,90 150x70)
            shows TEMPLATE_TEMP_SENSOR_VALUE_ONLY(m_instance := m_Instance.t_img_lmd_2_ramp)
        Frame (10,160 150x70)
            shows TEMPLATE_TEMP_SENSOR_VALUE_ONLY(m_instance := m_Instance.t_img_lmp_2_ramp)
        Frame (10,230 150x70)
            shows TEMPLATE_TEMP_SENSOR_VALUE_ONLY(m_instance := m_Instance.t_img_nd_2_ramp)
    Label (30,70 299x30), "Measured"
    Label (30,772 299x30), "Calculcated"
    Line (420,1142) (420,352)
END_VISUALIZATION

// HMI/VISUs/Subsystems/IMG/Components/VISU_HMI_IMG_VOTERS
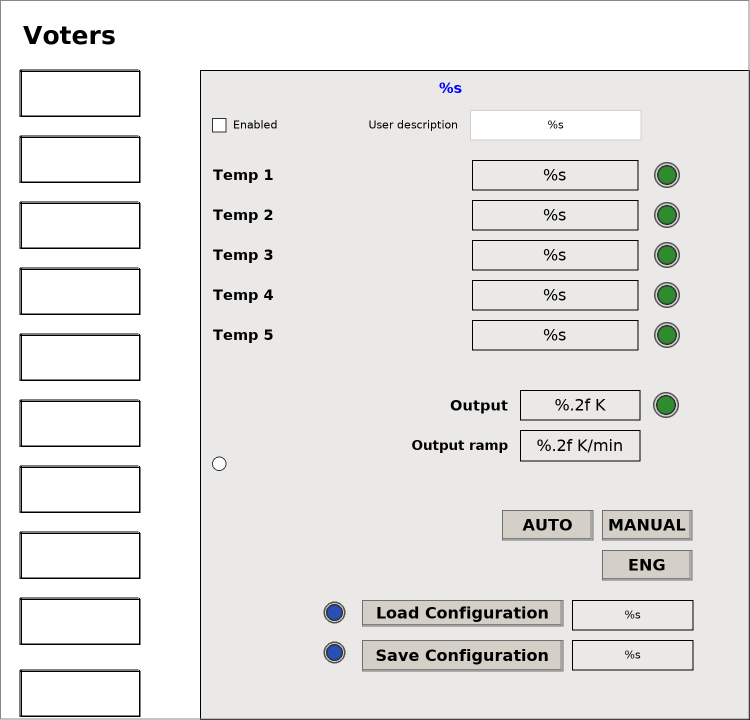
VISUALIZATION VISU_HMI_IMG_VOTERS  // 750x720
VAR_IN_OUT
    m_Instance : FB_METIS_VOTERS;
	m_Hmi : FB_HMI_IMG_VOTERS;
    m_temperatures : FB_METIS_TEMPERATURES;
END_VAR
    Rectangle (200,70 550x650)
    Frame (20,70 121x48)
        shows VISU_HMI_SUBSYSTEM_BUTTON(m_Hmi := m_Hmi.fbVoter1Button)
        OnMouseClick: execute { m_Hmi.eActiveTab := E_HMI_VOTER_TABS.VOTER_1; }
    Frame (20,136 121x48)
        shows VISU_HMI_SUBSYSTEM_BUTTON(m_Hmi := m_Hmi.fbVoter2Button)
        OnMouseClick: execute { m_Hmi.eActiveTab := E_HMI_VOTER_TABS.VOTER_2; }
    Frame (20,202 121x48)
        shows VISU_HMI_SUBSYSTEM_BUTTON(m_Hmi := m_Hmi.fbVoter3Button)
        OnMouseClick: execute { m_Hmi.eActiveTab := E_HMI_VOTER_TABS.VOTER_3; }
    Frame (20,268 121x48)
        shows VISU_HMI_SUBSYSTEM_BUTTON(m_Hmi := m_Hmi.fbVoter4Button)
        OnMouseClick: execute { m_Hmi.eActiveTab := E_HMI_VOTER_TABS.VOTER_4; }
    Frame (20,334 121x48)
        shows VISU_HMI_SUBSYSTEM_BUTTON(m_Hmi := m_Hmi.fbVoter5Button)
        OnMouseClick: execute { m_Hmi.eActiveTab := E_HMI_VOTER_TABS.VOTER_5; }
    Frame (20,400 121x48)
        shows VISU_HMI_SUBSYSTEM_BUTTON(m_Hmi := m_Hmi.fbVoter6Button)
        OnMouseClick: execute { m_Hmi.eActiveTab := E_HMI_VOTER_TABS.VOTER_6; }
    Frame (20,466 121x48)
        shows VISU_HMI_SUBSYSTEM_BUTTON(m_Hmi := m_Hmi.fbVoter7Button)
        OnMouseClick: execute { m_Hmi.eActiveTab := E_HMI_VOTER_TABS.VOTER_7; }
    Frame (20,532 121x48)
        shows VISU_HMI_SUBSYSTEM_BUTTON(m_Hmi := m_Hmi.fbVoter8Button)
        OnMouseClick: execute { m_Hmi.eActiveTab := E_HMI_VOTER_TABS.VOTER_8; }
    Frame (20,598 121x48)
        shows VISU_HMI_SUBSYSTEM_BUTTON(m_Hmi := m_Hmi.fbVoter9Button)
        OnMouseClick: execute { m_Hmi.eActiveTab := E_HMI_VOTER_TABS.VOTER_9; }
    Frame (20,670 121x48)
        shows VISU_HMI_SUBSYSTEM_BUTTON(m_Hmi := m_Hmi.fbVoter10Button)
        OnMouseClick: execute { m_Hmi.eActiveTab := E_HMI_VOTER_TABS.VOTER_10; }
    Frame (200,70 545x641), frame switch variable: m_Hmi.eActiveTab
        shows TEMPLATE_TEMPERATURE_VOTE(m_Instance := m_Instance.vote_img_1, m_all_temperatures_array := m_temperatures)
        shows TEMPLATE_TEMPERATURE_VOTE(m_Instance := m_Instance.vote_img_2, m_all_temperatures_array := m_temperatures)
        shows TEMPLATE_TEMPERATURE_VOTE(m_Instance := m_Instance.vote_img_3, m_all_temperatures_array := m_temperatures)
        shows TEMPLATE_TEMPERATURE_VOTE(m_Instance := m_Instance.vote_img_4, m_all_temperatures_array := m_temperatures)
        shows TEMPLATE_TEMPERATURE_VOTE(m_Instance := m_Instance.vote_img_5, m_all_temperatures_array := m_temperatures)
        shows TEMPLATE_TEMPERATURE_VOTE(m_Instance := m_Instance.vote_img_6, m_all_temperatures_array := m_temperatures)
        shows TEMPLATE_TEMPERATURE_VOTE(m_Instance := m_Instance.vote_img_7, m_all_temperatures_array := m_temperatures)
        shows TEMPLATE_TEMPERATURE_VOTE(m_Instance := m_Instance.vote_img_8, m_all_temperatures_array := m_temperatures)
        shows TEMPLATE_TEMPERATURE_VOTE(m_Instance := m_Instance.vote_img_9, m_all_temperatures_array := m_temperatures)
        shows TEMPLATE_TEMPERATURE_VOTE(m_Instance := m_Instance.vote_img_10, m_all_temperatures_array := m_temperatures)
    Label (20,20 411x30), "Voters"
END_VISUALIZATION

// HMI/VISUs/Subsystems/IMG/VISU_HMI_IMG
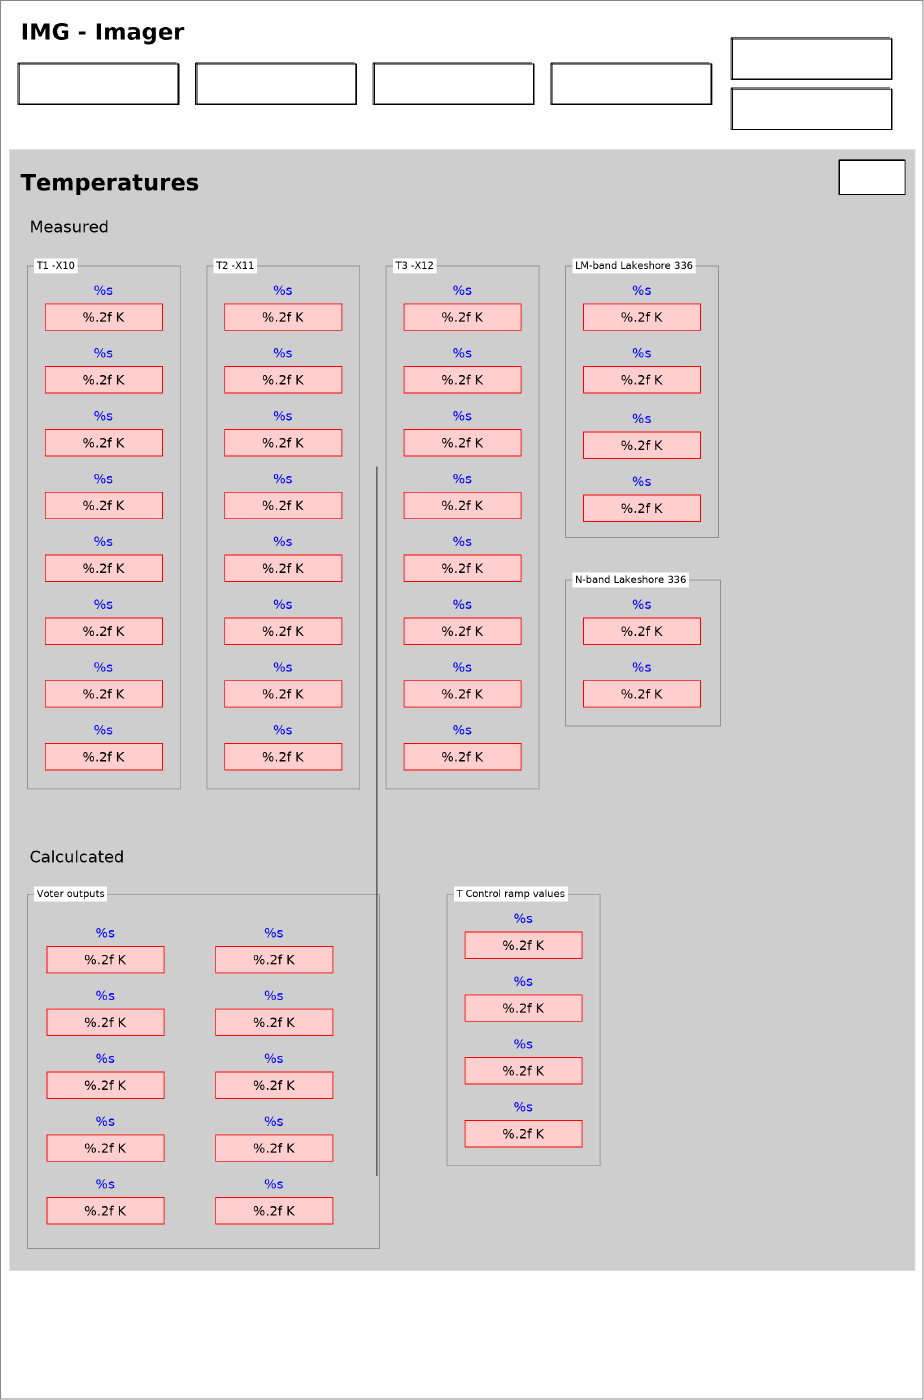
VISUALIZATION VISU_HMI_IMG  // 1030x1560
VAR_IN_OUT
	m_Temperatures : FB_METIS_TEMPERATURES;
    m_Voters : FB_METIS_VOTERS;
    m_Tctrl : FB_METIS_TCTRL;
    m_Heaters : FB_METIS_HEATERS;
    m_Lakeshores : FB_METIS_LAKESHORES;
    m_Hmi : FB_HMI_IMG;
END_VAR
    Frame (0,36 1021x1397)
        shows TEMPLATE_BACKGROUND_LEVEL_2()
    Label (20,20 671x30), "IMG - Imager"
    Frame (20,70 181x48)
        shows VISU_HMI_SUBSYSTEM_BUTTON(m_Hmi := m_Hmi.fbTemperaturesButton)
        OnMouseClick: execute { m_Hmi.eActiveTab := E_HMI_IMG_TABS.TEMPERATURES; }
    Frame (614,70 181x48)
        shows VISU_HMI_SUBSYSTEM_BUTTON(m_Hmi := m_Hmi.fbHeatersButton)
        OnMouseClick: execute { m_Hmi.eActiveTab := E_HMI_IMG_TABS.HEATERS; }
    Frame (218,70 181x48)
        shows VISU_HMI_SUBSYSTEM_BUTTON(m_Hmi := m_Hmi.fbVotersButton)
        OnMouseClick: execute { m_Hmi.eActiveTab := E_HMI_IMG_TABS.VOTERS; }
    Frame (416,70 181x48)
        shows VISU_HMI_SUBSYSTEM_BUTTON(m_Hmi := m_Hmi.fbTControlButton)
        OnMouseClick: execute { m_Hmi.eActiveTab := E_HMI_IMG_TABS.TCONTROL; }
    Group (815,42 181x104)
        Frame (0,0 181x48)
            shows VISU_HMI_SUBSYSTEM_BUTTON(m_Hmi := m_Hmi.fbLakeshoreLmButton)
            OnMouseClick: execute { m_Hmi.eActiveTab := E_HMI_IMG_TABS.LAKESHORE_LM_DET; }
        Frame (0,56 181x48)
            shows VISU_HMI_SUBSYSTEM_BUTTON(m_Hmi := m_Hmi.fbLakeshoreNButton)
            OnMouseClick: execute { m_Hmi.eActiveTab := E_HMI_IMG_TABS.LAKESHORE_N_DET; }
    Frame (0,168 1017x1250), frame switch variable: m_Hmi.eActiveTab
        shows VISU_HMI_IMG_TEMPERATURES(m_Instance := m_Temperatures)
        shows VISU_HMI_IMG_VOTERS(m_Instance := m_Voters, m_Hmi := m_Hmi.fbVoters, m_temperatures := m_Temperatures)
        shows VISU_HMI_IMG_TC(m_Instance := m_Tctrl, m_Hmi := m_Hmi.fbTControl, m_temp := m_Temperatures)
        shows VISU_HMI_IMG_HEATERS(m_Instance := m_Heaters, m_Hmi := m_Hmi.fbHeaters)
        shows GUI_TEMPLATE_LAKESHORE_336_TCP(m_Instance := m_Lakeshores.ls_img_lm)
        shows GUI_TEMPLATE_LAKESHORE_336_TCP(m_Instance := m_Lakeshores.ls_img_n)
    Frame (935,178 75x40)
        shows VISU_HMI_SUBSYSTEM_BUTTON(m_Hmi := PRG_HMI.fbBackButton)
        OnMouseClick: execute { PRG_HMI.eActiveTab := PRG_HMI.ePreviousTab; }
END_VISUALIZATION

// HMI/VISUs/Subsystems/LMS/VISU_HMI_LMS
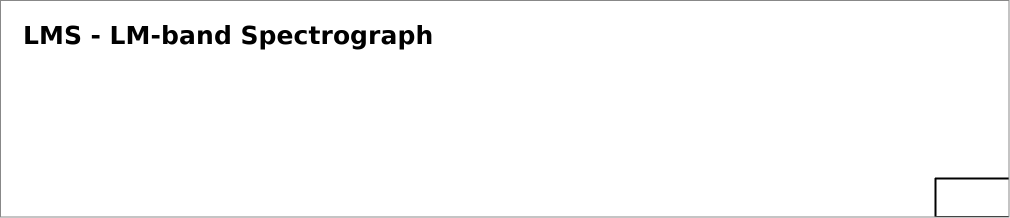
VISUALIZATION VISU_HMI_LMS  // 1010x218
    Label (20,20 671x30), "LMS - LM-band Spectrograph"
    Frame (935,178 75x40)
        shows VISU_HMI_SUBSYSTEM_BUTTON(m_Hmi := PRG_HMI.fbBackButton)
        OnMouseClick: execute { PRG_HMI.eActiveTab := PRG_HMI.ePreviousTab; }
END_VISUALIZATION

// HMI/VISUs/Subsystems/SCA/Components/VISU_HMI_SCA_HEATERS
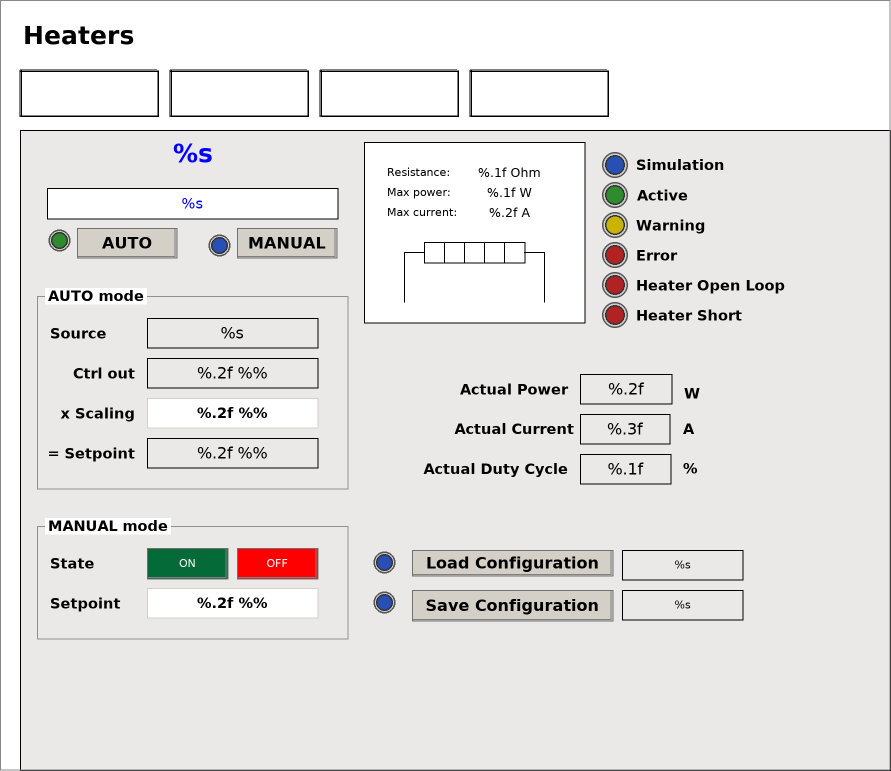
VISUALIZATION VISU_HMI_SCA_HEATERS  // 891x771
VAR_IN_OUT
	m_Instance : FB_METIS_HEATERS;
    m_Hmi : FB_HMI_SCA_HEATERS;
END_VAR
    Rectangle (20,130 871x641)
    Label (20,20 411x30), "Heaters"
    Frame (20,130 800x550), frame switch variable: m_Hmi.eActiveTab
        shows TEMPLATE_METIS_HEATER(m_instance := m_Instance.h_sca_wuh_1)
        shows TEMPLATE_METIS_HEATER(m_instance := m_Instance.h_sca_wuh_2)
        shows TEMPLATE_METIS_HEATER(m_instance := m_Instance.h_sca_det_2)
        shows TEMPLATE_METIS_HEATER(m_instance := m_Instance.h_sca_dhs_2)
        shows METIS_Cryo_PLC.TEMPLATE_METIS_CTRL_DT670(m_temp := m_temp)
        shows METIS_Cryo_PLC.TEMPLATE_METIS_HEATER(m_instance := m_Instance.h_img_nd_2)
        p8630679: tcontrol.tc_img_wuh_1
        p371692913: tcontrol.vote_img_wuh_1
        p2286783886: temperatures
    Frame (20,70 140x48)
        shows VISU_HMI_SUBSYSTEM_BUTTON(m_Hmi := m_Hmi.h_sca_wuh_1_button)
        OnMouseClick: execute { m_Hmi.eActiveTab := E_HMI_SCA_HEATER_TABS.H_SCA_WUH_1; }
    Frame (170,70 140x48)
        shows VISU_HMI_SUBSYSTEM_BUTTON(m_Hmi := m_Hmi.h_sca_wuh_2_button)
        OnMouseClick: execute { m_Hmi.eActiveTab := E_HMI_SCA_HEATER_TABS.H_SCA_WUH_2; }
    Frame (320,70 140x48)
        shows VISU_HMI_SUBSYSTEM_BUTTON(m_Hmi := m_Hmi.h_sca_det_2_button)
        OnMouseClick: execute { m_Hmi.eActiveTab := E_HMI_SCA_HEATER_TABS.H_SCA_DET_2; }
    Frame (470,70 140x48)
        shows VISU_HMI_SUBSYSTEM_BUTTON(m_Hmi := m_Hmi.h_sca_dhs_2_button)
        OnMouseClick: execute { m_Hmi.eActiveTab := E_HMI_SCA_HEATER_TABS.H_SCA_DHS_2; }
END_VISUALIZATION

// HMI/VISUs/Subsystems/SCA/Components/VISU_HMI_SCA_TC
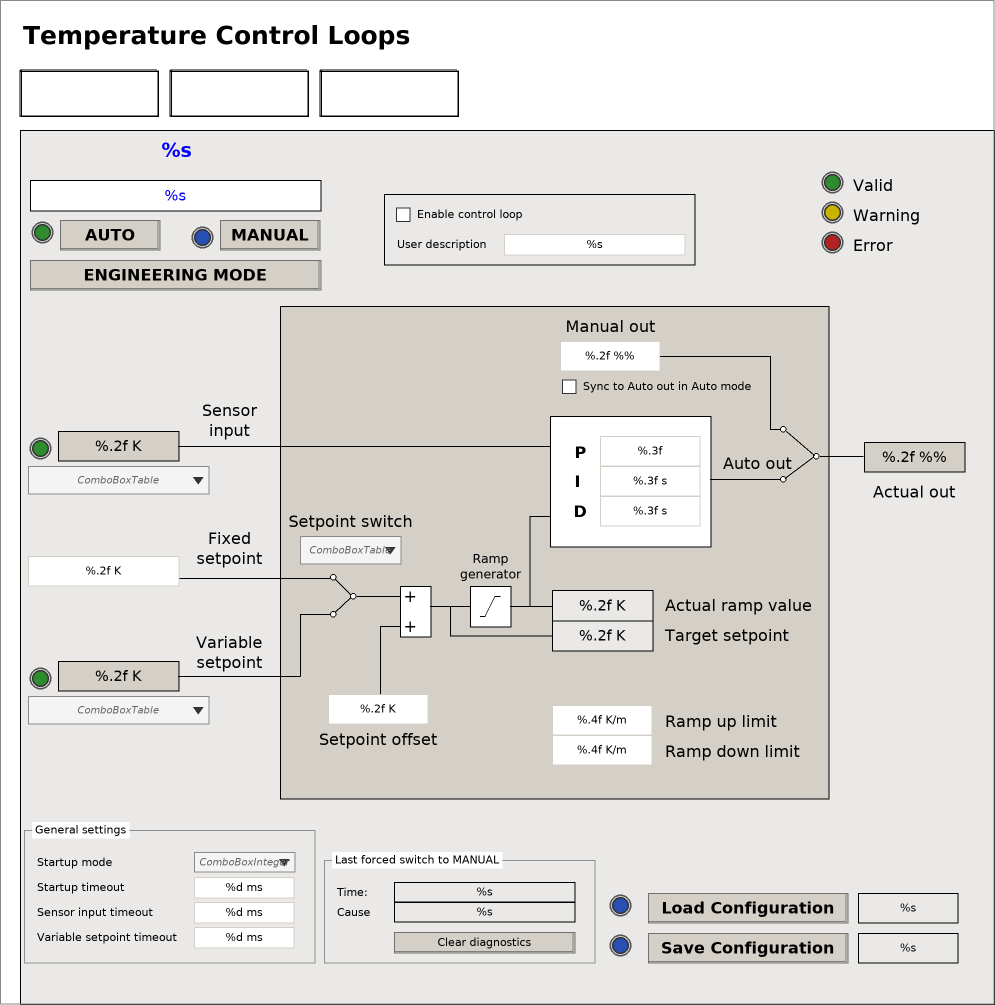
VISUALIZATION VISU_HMI_SCA_TC  // 995x1005
VAR_IN_OUT
    m_Instance : FB_METIS_TCTRL;
    m_Hmi : FB_HMI_SCA_TCTRL;
    m_temp : FB_METIS_TEMPERATURES;
END_VAR
    Rectangle (20,130 975x875)
    Label (20,20 411x30), "Temperature Control Loops"
    Frame (20,130 975x875), frame switch variable: m_Hmi.eActiveTab
        shows TEMPLATE_METIS_CTRL_TEMPERATURE(m_instance := m_Instance.tc_sca_wuh, m_temp := m_temp)
        shows TEMPLATE_METIS_CTRL_TEMPERATURE(m_instance := m_Instance.tc_sca_det_2, m_temp := m_temp)
        shows TEMPLATE_METIS_CTRL_TEMPERATURE(m_instance := m_Instance.tc_sca_dhs_2, m_temp := m_temp)
        shows METIS_Cryo_PLC.TEMPLATE_METIS_CTRL_DT670(m_instance := m_Instance.tc_img_nd_2, m_temp := m_temp)
        shows METIS_Cryo_PLC.TEMPLATE_METIS_CTRL_DT670(m_temp := m_temp)
        shows TEMPLATE_METIS_CTRL_TEMPERATURE(m_instance := m_Instance.tc_sca_dhs_2, m_temp := m_temp)
        p8630679: tcontrol.tc_img_wuh_1
        p371692913: tcontrol.vote_img_wuh_1
        p2286783886: temperatures
    Frame (20,70 140x48)
        shows VISU_HMI_SUBSYSTEM_BUTTON(m_Hmi := m_Hmi.tc_sca_wuh_button)
        OnMouseClick: execute { m_Hmi.eActiveTab := E_HMI_SCA_TC_TABS.TC_SCA_WUH; }
    Frame (170,70 140x48)
        shows VISU_HMI_SUBSYSTEM_BUTTON(m_Hmi := m_Hmi.tc_sca_det_2_button)
        OnMouseClick: execute { m_Hmi.eActiveTab := E_HMI_SCA_TC_TABS.TC_SCA_DET_2; }
    Frame (320,70 140x48)
        shows VISU_HMI_SUBSYSTEM_BUTTON(m_Hmi := m_Hmi.tc_sca_dhs_2_button)
        OnMouseClick: execute { m_Hmi.eActiveTab := E_HMI_SCA_TC_TABS.TC_SCA_DHS_2; }
END_VISUALIZATION

// HMI/VISUs/Subsystems/SCA/Components/VISU_HMI_SCA_TEMPERATURES
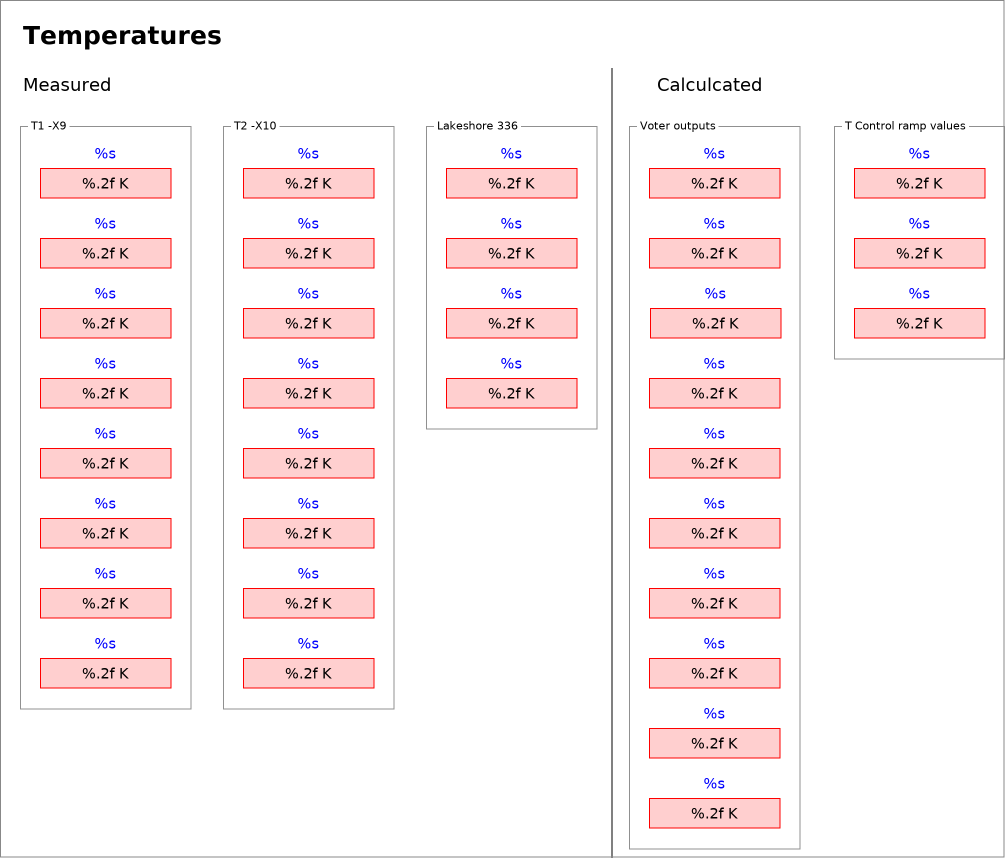
VISUALIZATION VISU_HMI_SCA_TEMPERATURES  // 1005x858
VAR_IN_OUT
	m_Instance : FB_METIS_TEMPERATURES;
END_VAR
    Label (20,20 299x30), "Temperatures"
    GroupBox (20,118 171x591), "T1 -X9"
        Frame (10,20 150x70)
            shows TEMPLATE_TEMP_SENSOR_VALUE_ONLY(m_instance := m_Instance.t_sca_fw_1)
        Frame (10,90 150x70)
            shows TEMPLATE_TEMP_SENSOR_VALUE_ONLY(m_instance := m_Instance.t_sca_fw_2)
        Frame (10,160 150x70)
            shows TEMPLATE_TEMP_SENSOR_VALUE_ONLY(m_instance := m_Instance.t_sca_lu_1)
        Frame (10,230 150x70)
            shows TEMPLATE_TEMP_SENSOR_VALUE_ONLY(m_instance := m_Instance.t_sca_fm)
        Frame (10,300 150x70)
            shows TEMPLATE_TEMP_SENSOR_VALUE_ONLY(m_instance := m_Instance.t_sca_fs)
        Frame (10,370 150x70)
            shows TEMPLATE_TEMP_SENSOR_VALUE_ONLY(m_instance := m_Instance.t_sca_lu_2)
        Frame (10,440 150x70)
            shows TEMPLATE_TEMP_SENSOR_VALUE_ONLY(m_instance := m_Instance.t_sca_mod)
        Frame (10,510 150x70)
            shows TEMPLATE_TEMP_SENSOR_VALUE_ONLY(m_instance := m_Instance.t_sca_pyr)
    GroupBox (223,118 171x591), "T2 -X10"
        Frame (10,20 150x70)
            shows TEMPLATE_TEMP_SENSOR_VALUE_ONLY(m_instance := m_Instance.t_sca_h_1)
        Frame (10,90 150x70)
            shows TEMPLATE_TEMP_SENSOR_VALUE_ONLY(m_instance := m_Instance.t_sca_if_1)
        Frame (10,160 150x70)
            shows TEMPLATE_TEMP_SENSOR_VALUE_ONLY(m_instance := m_Instance.t_sca_if_2)
        Frame (10,230 150x70)
            shows TEMPLATE_TEMP_SENSOR_VALUE_ONLY(m_instance := m_Instance.t_sca_lu_3)
        Frame (10,300 150x70)
            shows TEMPLATE_TEMP_SENSOR_VALUE_ONLY(m_instance := m_Instance.t_sca_bp_1)
        Frame (10,370 150x70)
            shows TEMPLATE_TEMP_SENSOR_VALUE_ONLY(m_instance := m_Instance.t_sca_bp_2)
        Frame (10,440 150x70)
            shows TEMPLATE_TEMP_SENSOR_VALUE_ONLY(m_instance := m_Instance.t_sca_bp_3)
        Frame (10,510 150x70)
            shows TEMPLATE_TEMP_SENSOR_VALUE_ONLY(m_instance := m_Instance.t_sca_h_2)
    GroupBox (426,118 171x311), "Lakeshore 336"
        Frame (10,20 150x70)
            shows TEMPLATE_TEMP_SENSOR_VALUE_ONLY(m_instance := m_Instance.t_sca_det_1)
        Frame (10,90 150x70)
            shows TEMPLATE_TEMP_SENSOR_VALUE_ONLY(m_instance := m_Instance.t_sca_det_2)
        Frame (10,160 150x70)
            shows TEMPLATE_TEMP_SENSOR_VALUE_ONLY(m_instance := m_Instance.t_sca_dhs_1)
        Frame (10,230 150x70)
            shows TEMPLATE_TEMP_SENSOR_VALUE_ONLY(m_instance := m_Instance.t_sca_dhs_2)
    GroupBox (629,118 171x731), "Voter outputs"
        Frame (10,20 150x70)
            shows TEMPLATE_TEMP_SENSOR_VALUE_ONLY(m_instance := m_Instance.t_sca_vot_1)
        Frame (10,90 150x70)
            shows TEMPLATE_TEMP_SENSOR_VALUE_ONLY(m_instance := m_Instance.t_sca_vot_2)
        Frame (10,230 150x70)
            shows TEMPLATE_TEMP_SENSOR_VALUE_ONLY(m_instance := m_Instance.t_sca_vot_4)
        Frame (10,300 150x70)
            shows TEMPLATE_TEMP_SENSOR_VALUE_ONLY(m_instance := m_Instance.t_sca_vot_5)
        Frame (10,370 150x70)
            shows TEMPLATE_TEMP_SENSOR_VALUE_ONLY(m_instance := m_Instance.t_sca_vot_6)
        Frame (10,440 150x70)
            shows TEMPLATE_TEMP_SENSOR_VALUE_ONLY(m_instance := m_Instance.t_sca_vot_7)
        Frame (10,510 150x70)
            shows TEMPLATE_TEMP_SENSOR_VALUE_ONLY(m_instance := m_Instance.t_sca_vot_8)
        Frame (10,580 150x70)
            shows TEMPLATE_TEMP_SENSOR_VALUE_ONLY(m_instance := m_Instance.t_sca_vot_9)
        Frame (10,650 150x70)
            shows TEMPLATE_TEMP_SENSOR_VALUE_ONLY(m_instance := m_Instance.t_sca_vot_10)
        Frame (11,160 150x70)
            shows TEMPLATE_TEMP_SENSOR_VALUE_ONLY(m_instance := m_Instance.t_sca_vot_3)
    GroupBox (834,118 171x241), "T Control ramp values"
        Frame (10,20 150x70)
            shows TEMPLATE_TEMP_SENSOR_VALUE_ONLY(m_instance := m_Instance.t_sca_wuh_ramp)
        Frame (10,90 150x70)
            shows TEMPLATE_TEMP_SENSOR_VALUE_ONLY(m_instance := m_Instance.t_sca_det_2_ramp)
        Frame (10,160 150x70)
            shows TEMPLATE_TEMP_SENSOR_VALUE_ONLY(m_instance := m_Instance.t_sca_dhs_2_ramp)
    Label (20,70 299x30), "Measured"
    Label (654,70 299x30), "Calculcated"
    Line (612,858) (612,68)
END_VISUALIZATION

// HMI/VISUs/Subsystems/SCA/Components/VISU_HMI_SCA_VOTERS
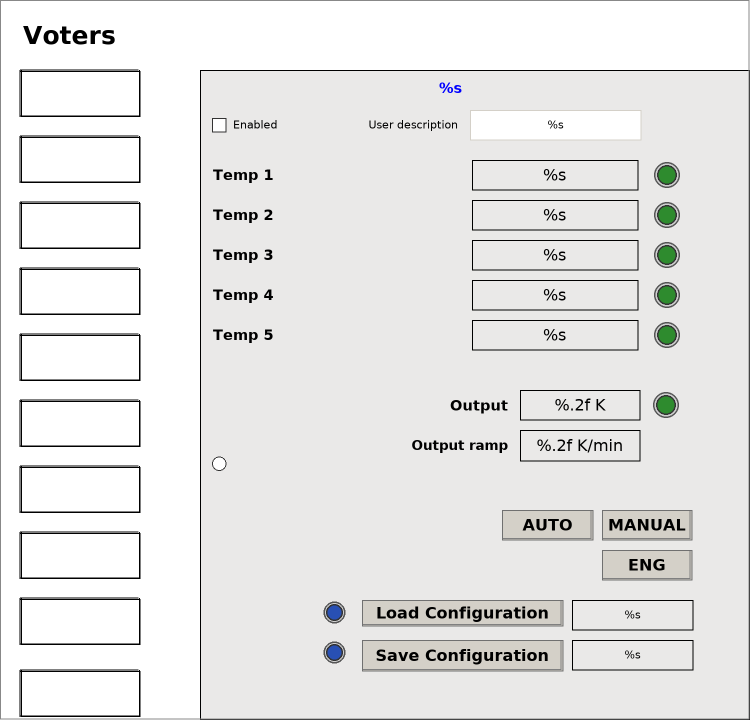
VISUALIZATION VISU_HMI_SCA_VOTERS  // 750x720
VAR_IN_OUT
    m_Instance : FB_METIS_VOTERS;
	m_Hmi : FB_HMI_SCA_VOTERS;
    m_temperatures : FB_METIS_TEMPERATURES;
END_VAR
    Rectangle (200,70 550x650)
    Frame (20,70 121x48)
        shows VISU_HMI_SUBSYSTEM_BUTTON(m_Hmi := m_Hmi.fbVoter1Button)
        OnMouseClick: execute { m_Hmi.eActiveTab := E_HMI_VOTER_TABS.VOTER_1; }
    Frame (20,136 121x48)
        shows VISU_HMI_SUBSYSTEM_BUTTON(m_Hmi := m_Hmi.fbVoter2Button)
        OnMouseClick: execute { m_Hmi.eActiveTab := E_HMI_VOTER_TABS.VOTER_2; }
    Frame (20,202 121x48)
        shows VISU_HMI_SUBSYSTEM_BUTTON(m_Hmi := m_Hmi.fbVoter3Button)
        OnMouseClick: execute { m_Hmi.eActiveTab := E_HMI_VOTER_TABS.VOTER_3; }
    Frame (20,268 121x48)
        shows VISU_HMI_SUBSYSTEM_BUTTON(m_Hmi := m_Hmi.fbVoter4Button)
        OnMouseClick: execute { m_Hmi.eActiveTab := E_HMI_VOTER_TABS.VOTER_4; }
    Frame (20,334 121x48)
        shows VISU_HMI_SUBSYSTEM_BUTTON(m_Hmi := m_Hmi.fbVoter5Button)
        OnMouseClick: execute { m_Hmi.eActiveTab := E_HMI_VOTER_TABS.VOTER_5; }
    Frame (20,400 121x48)
        shows VISU_HMI_SUBSYSTEM_BUTTON(m_Hmi := m_Hmi.fbVoter6Button)
        OnMouseClick: execute { m_Hmi.eActiveTab := E_HMI_VOTER_TABS.VOTER_6; }
    Frame (20,466 121x48)
        shows VISU_HMI_SUBSYSTEM_BUTTON(m_Hmi := m_Hmi.fbVoter7Button)
        OnMouseClick: execute { m_Hmi.eActiveTab := E_HMI_VOTER_TABS.VOTER_7; }
    Frame (20,532 121x48)
        shows VISU_HMI_SUBSYSTEM_BUTTON(m_Hmi := m_Hmi.fbVoter8Button)
        OnMouseClick: execute { m_Hmi.eActiveTab := E_HMI_VOTER_TABS.VOTER_8; }
    Frame (20,598 121x48)
        shows VISU_HMI_SUBSYSTEM_BUTTON(m_Hmi := m_Hmi.fbVoter9Button)
        OnMouseClick: execute { m_Hmi.eActiveTab := E_HMI_VOTER_TABS.VOTER_9; }
    Frame (20,670 121x48)
        shows VISU_HMI_SUBSYSTEM_BUTTON(m_Hmi := m_Hmi.fbVoter10Button)
        OnMouseClick: execute { m_Hmi.eActiveTab := E_HMI_VOTER_TABS.VOTER_10; }
    Frame (200,70 550x641), frame switch variable: m_Hmi.eActiveTab
        shows TEMPLATE_TEMPERATURE_VOTE(m_Instance := m_Instance.vote_sca_1, m_all_temperatures_array := m_temperatures)
        shows TEMPLATE_TEMPERATURE_VOTE(m_Instance := m_Instance.vote_sca_2, m_all_temperatures_array := m_temperatures)
        shows TEMPLATE_TEMPERATURE_VOTE(m_Instance := m_Instance.vote_sca_3, m_all_temperatures_array := m_temperatures)
        shows TEMPLATE_TEMPERATURE_VOTE(m_Instance := m_Instance.vote_sca_4, m_all_temperatures_array := m_temperatures)
        shows TEMPLATE_TEMPERATURE_VOTE(m_Instance := m_Instance.vote_sca_5, m_all_temperatures_array := m_temperatures)
        shows TEMPLATE_TEMPERATURE_VOTE(m_Instance := m_Instance.vote_sca_6, m_all_temperatures_array := m_temperatures)
        shows TEMPLATE_TEMPERATURE_VOTE(m_Instance := m_Instance.vote_sca_7, m_all_temperatures_array := m_temperatures)
        shows TEMPLATE_TEMPERATURE_VOTE(m_Instance := m_Instance.vote_sca_8, m_all_temperatures_array := m_temperatures)
        shows TEMPLATE_TEMPERATURE_VOTE(m_Instance := m_Instance.vote_sca_9, m_all_temperatures_array := m_temperatures)
        shows TEMPLATE_TEMPERATURE_VOTE(m_Instance := m_Instance.vote_sca_10, m_all_temperatures_array := m_temperatures)
    Label (20,20 411x30), "Voters"
END_VISUALIZATION

// HMI/VISUs/Subsystems/SCA/VISU_HMI_SCA
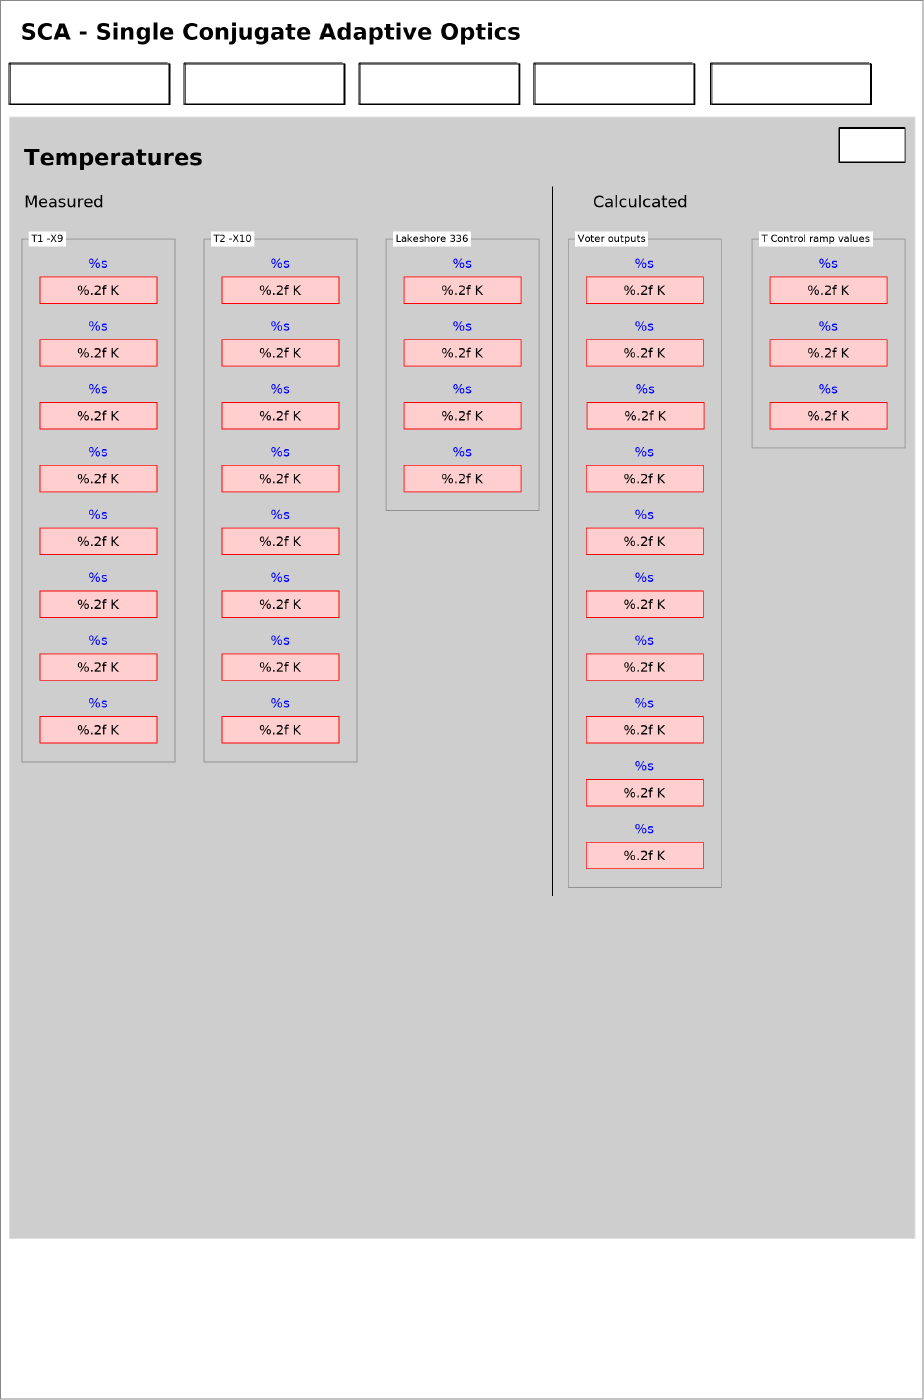
VISUALIZATION VISU_HMI_SCA  // 1030x1560
VAR_IN_OUT
	m_Temperatures : FB_METIS_TEMPERATURES;
    m_Voters : FB_METIS_VOTERS;
    m_Tctrl : FB_METIS_TCTRL;
    m_Heaters : FB_METIS_HEATERS;
    m_Lakeshores : FB_METIS_LAKESHORES;
    m_Hmi : FB_HMI_SCA;
END_VAR
    Frame (0,0 1021x1425)
        shows TEMPLATE_BACKGROUND_LEVEL_2()
    Label (20,20 671x30), "SCA - Single Conjugate Adaptive Optics"
    Frame (10,70 181x48)
        shows VISU_HMI_SUBSYSTEM_BUTTON(m_Hmi := m_Hmi.fbTemperaturesButton)
        OnMouseClick: execute { m_Hmi.eActiveTab := E_HMI_SCA_TABS.TEMPERATURES; }
    Frame (595,70 181x48)
        shows VISU_HMI_SUBSYSTEM_BUTTON(m_Hmi := m_Hmi.fbHeatersButton)
        OnMouseClick: execute { m_Hmi.eActiveTab := E_HMI_SCA_TABS.HEATERS; }
    Frame (205,70 181x48)
        shows VISU_HMI_SUBSYSTEM_BUTTON(m_Hmi := m_Hmi.fbVotersButton)
        OnMouseClick: execute { m_Hmi.eActiveTab := E_HMI_SCA_TABS.VOTERS; }
    Frame (400,70 181x48)
        shows VISU_HMI_SUBSYSTEM_BUTTON(m_Hmi := m_Hmi.fbTControlButton)
        OnMouseClick: execute { m_Hmi.eActiveTab := E_HMI_SCA_TABS.TCONTROL; }
    Frame (792,70 181x48)
        shows VISU_HMI_SUBSYSTEM_BUTTON(m_Hmi := m_Hmi.fbLakeshoreButton)
        OnMouseClick: execute { m_Hmi.eActiveTab := E_HMI_SCA_TABS.LAKESHORE_DET; }
    Frame (4,140 1005x871), frame switch variable: m_Hmi.eActiveTab
        shows VISU_HMI_SCA_TEMPERATURES(m_Instance := m_Temperatures)
        shows VISU_HMI_SCA_VOTERS(m_Instance := m_Voters, m_Hmi := m_Hmi.fbVoters, m_temperatures := m_Temperatures)
        shows VISU_HMI_SCA_TC(m_Instance := m_Tctrl, m_Hmi := m_Hmi.fbTControl, m_temp := m_Temperatures)
        shows VISU_HMI_SCA_HEATERS(m_Instance := m_Heaters, m_Hmi := m_Hmi.fbHeaters)
        shows GUI_TEMPLATE_LAKESHORE_336_TCP(m_Instance := m_Lakeshores.ls_sca)
        p2394187509: m_Lakeshores.ls_img_n
    Frame (935,142 75x40)
        shows VISU_HMI_SUBSYSTEM_BUTTON(m_Hmi := PRG_HMI.fbBackButton)
        OnMouseClick: execute { PRG_HMI.eActiveTab := PRG_HMI.ePreviousTab; }
END_VISUALIZATION

// HMI/VISUs/Templates/ARCHIVED_TEMPLATE_MAIN_FSM_1
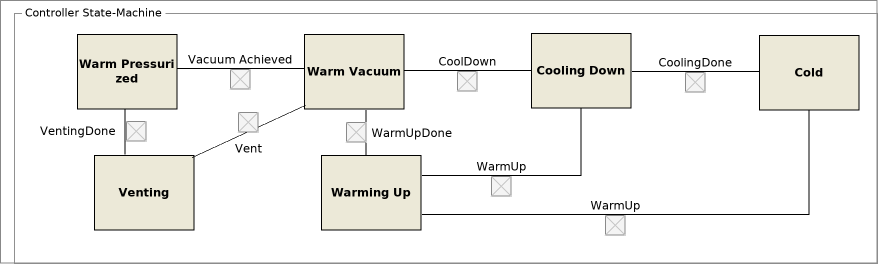
VISUALIZATION ARCHIVED_TEMPLATE_MAIN_FSM_1  // 878x264
VAR_IN_OUT
	m_instance:	FB_METIS_CRYO_CTRL;
END_VAR
    GroupBox (14,5 864x259), "Controller State-Machine"
    Group (33,33 826x202)
        RoundedRectangle (498,0 100x75), "Cooling Down", colour toggle: m_instance.stat.nState = E_METIS_CRYO_CTRL_STATE.COOLING_DOWN
        RoundedRectangle (288,122 100x75), "Warming Up", colour toggle: m_instance.stat.nState = E_METIS_CRYO_CTRL_STATE.WARMING_UP
        RoundedRectangle (726,2 100x75), "Cold", colour toggle: m_instance.stat.nState = E_METIS_CRYO_CTRL_STATE.COLD
        RoundedRectangle (61,122 100x75), "Venting", colour toggle: m_instance.stat.nState = E_METIS_CRYO_CTRL_STATE.VENTING
        RoundedRectangle (44,1 100x75), "Warm Pressurized", colour toggle: m_instance.stat.nState = E_METIS_CRYO_CTRL_STATE.WARM_PRESS
        RoundedRectangle (271,1 100x75), "Warm Vacuum", colour toggle: m_instance.stat.nState = E_METIS_CRYO_CTRL_STATE.WARM_VACUUM
        Line (144,35) (271,35), "Vacuum Achieved"
        Line (371,37) (498,37), "CoolDown", colour toggle: m_instance.ctrl.bSafe_Cool_Down
        Line (599,38) (726,38), "CoolingDone"
        Line (389,181) (776,181), "WarmUp", colour toggle: m_instance.ctrl.bSafe_Warm_Up AND m_instance.stat.nState = E_METIS_CRYO_CTRL_STATE.COLD
        Line (389,142) (548,142), "WarmUp", colour toggle: m_instance.ctrl.bSafe_Warm_Up AND m_instance.stat.nState = E_METIS_CRYO_CTRL_STATE.COOLING_DOWN
        Line (776,181) (776,77), colour toggle: m_instance.ctrl.bSafe_Warm_Up AND m_instance.stat.nState = E_METIS_CRYO_CTRL_STATE.COLD
        Line (548,142) (548,75), colour toggle: m_instance.ctrl.bSafe_Warm_Up AND m_instance.stat.nState = E_METIS_CRYO_CTRL_STATE.COOLING_DOWN
        Line (333,122) (333,77)
        Line (92,121) (92,76)
        Rectangle (334,85 90x30), "WarmUpDone"
        Rectangle (0,83 90x30), "VentingDone"
        Line (159,124) (272,72), "Vent", colour toggle: m_instance.ctrl.bSafe_Cool_Down AND m_instance.stat.nState = E_METIS_CRYO_CTRL_STATE.WARM_VACUUM
        Image (652,39 20x20), image: VisuSymbols.Symbols.ArrowForward
        Image (424,38 20x20), image: VisuSymbols.Symbols.ArrowForward
        Image (197,36 20x20), image: VisuSymbols.Symbols.ArrowForward
        Image (572,182 20x20), image: VisuSymbols.Symbols.ArrowBack
        Image (458,143 20x20), image: VisuSymbols.Symbols.ArrowBack
        Image (205,79 20x20), angle 335, image: VisuSymbols.Symbols.ArrowBack
        Image (93,88 20x20), angle 90, image: VisuSymbols.Symbols.ArrowBack
        Image (313,89 20x20), angle 90, image: VisuSymbols.Symbols.ArrowBack
END_VISUALIZATION

// HMI/VISUs/Templates/GUI_EVAC_BRANCH_A_1
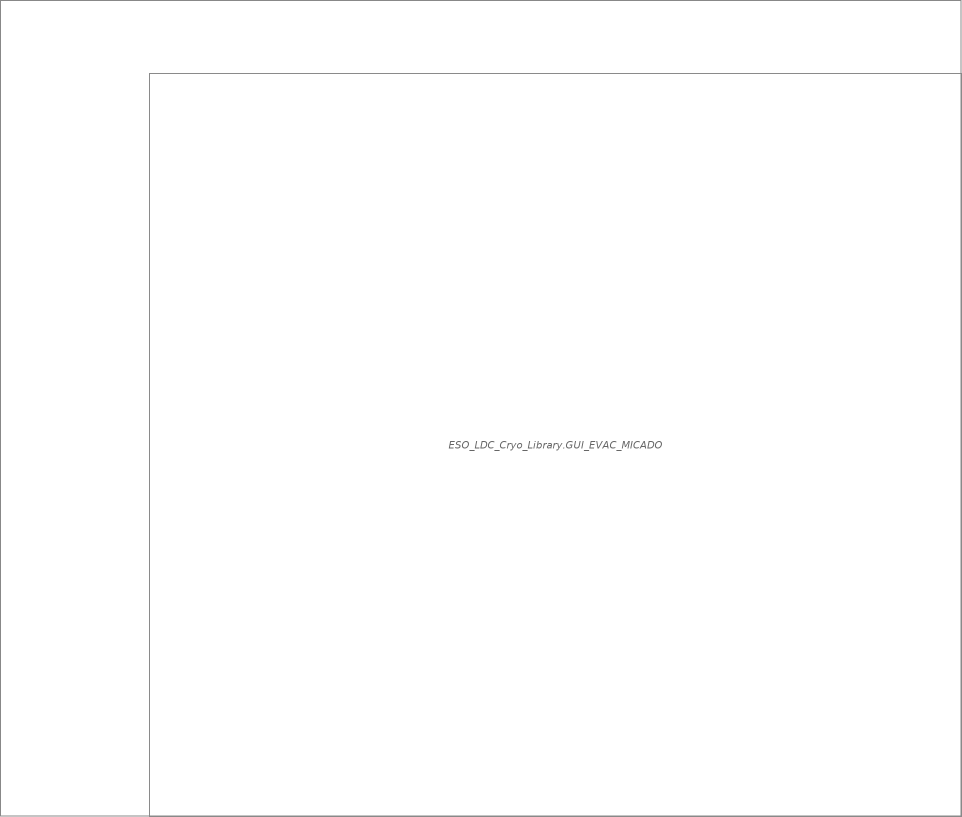
VISUALIZATION GUI_EVAC_BRANCH_A_1  // 962x817
    Frame (149,73 813x744)
        shows ESO_LDC_Cryo_Library.GUI_EVAC_MICADO()
END_VISUALIZATION

// HMI/VISUs/Templates/GUI_Events
VISUALIZATION GUI_Events  // 2x2
END_VISUALIZATION

// HMI/VISUs/Templates/GUI_RP_PUMPS
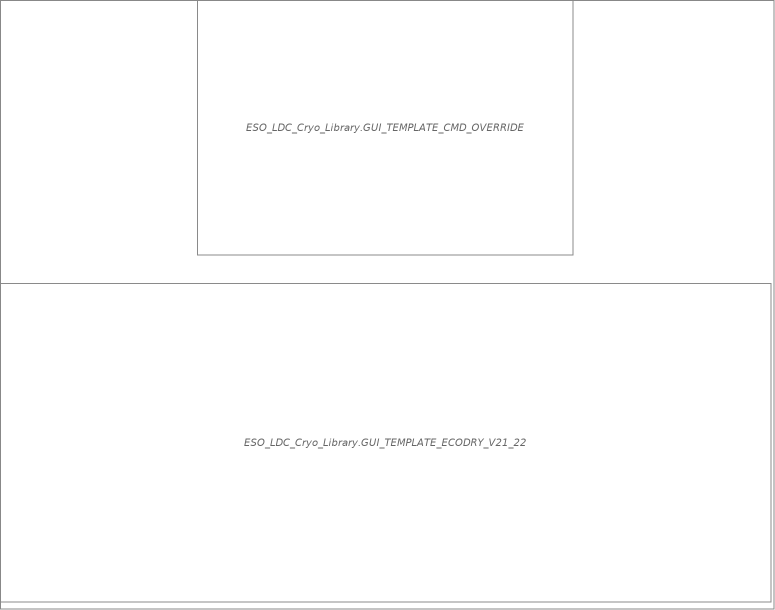
VISUALIZATION GUI_RP_PUMPS  // 775x610
    Frame (0,283 771x319)
        shows ESO_LDC_Cryo_Library.GUI_TEMPLATE_ECODRY_V21_22(m_Instance := MAIN.met_cryo_ctrl.met_evac.evac_branch_a.rp, m_bEnable := MAIN.met_cryo_ctrl.met_evac.evac_branch_a.rp.in_bEnable)
    Frame (197,0 376x255)
        shows ESO_LDC_Cryo_Library.GUI_TEMPLATE_CMD_OVERRIDE(m_Cmd := MAIN.met_cryo_ctrl.met_evac.evac_branch_a.cor_rp)
END_VISUALIZATION

// HMI/VISUs/Templates/GUI_TEMPLATE_LAKESHORE_336_TCP
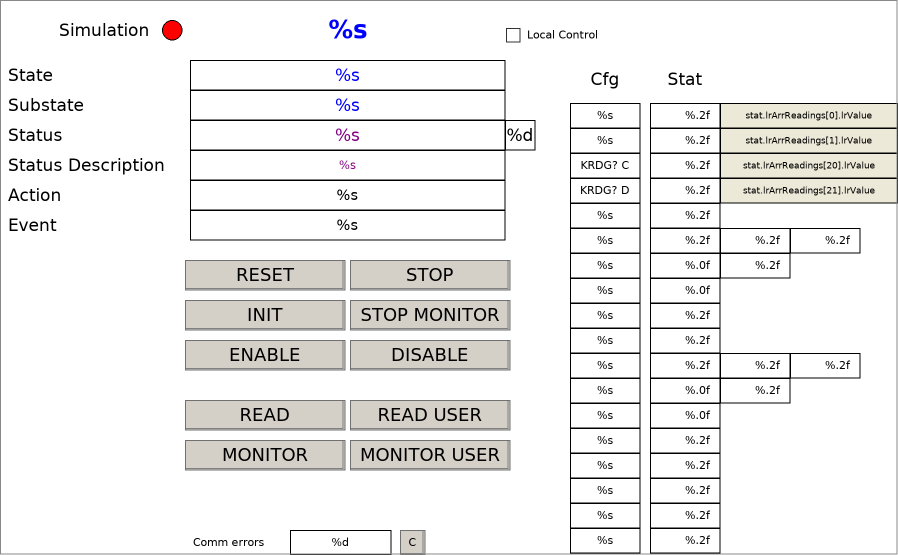
VISUALIZATION GUI_TEMPLATE_LAKESHORE_336_TCP  // 898x555
VAR_IN_OUT
	m_Instance:	FB_METIS_LAKESHORE_336_TCP;
END_VAR
    Rectangle (190,60 315x30), "%s", text variable: m_Instance.stat.sState
    Rectangle (190,90 315x30), "%s", text variable: m_Instance.stat.sSubstate
    Button (185,260 160x30), "RESET", input disabled if: (m_Instance.stat.bLocal = FALSE) <> 0
        OnMouseClick: execute { m_Instance.ctrl.nCommand := E_RS_COMMAND.RESET; m_Instance.ctrl.bExecute := TRUE; }
    Button (185,300 160x30), "INIT", input disabled if: (m_Instance.stat.bLocal = FALSE) <> 0
        OnMouseClick: execute { m_Instance.ctrl.nCommand := E_RS_COMMAND.INIT; m_Instance.ctrl.bExecute := TRUE; }
    Button (350,260 160x30), "STOP", input disabled if: (m_Instance.stat.bLocal = FALSE) <> 0
        OnMouseClick: execute { m_Instance.ctrl.nCommand := E_RS_COMMAND.STOP; m_Instance.ctrl.bExecute := TRUE; }
    Button (185,340 160x30), "ENABLE", input disabled if: (m_Instance.stat.bLocal = FALSE) <> 0
        OnMouseClick: execute { m_Instance.ctrl.nCommand := E_RS_COMMAND.ENABLE; m_Instance.ctrl.bExecute := TRUE; }
    Button (350,340 160x30), "DISABLE", input disabled if: (m_Instance.stat.bLocal = FALSE) <> 0
        OnMouseClick: execute { m_Instance.ctrl.nCommand := E_RS_COMMAND.DISABLE; m_Instance.ctrl.bExecute := TRUE; }
    Rectangle (5,60 180x30), "State"
    Rectangle (5,90 180x30), "Substate"
    Rectangle (190,120 315x30), "%s", text variable: m_Instance.stat.sStatus
    Rectangle (190,150 315x30), "%s", text variable: m_Instance.stat.sErrorText
    Rectangle (5,120 180x30), "Status"
    Rectangle (5,150 180x30), "Status Description"
    Rectangle (190,180 315x30), "%s", text variable: m_Instance.stat.sActionDesc
    Rectangle (190,210 315x30), "%s", text variable: m_Instance.stat.sEventDesc
    Rectangle (5,180 180x30), "Action"
    Rectangle (5,210 180x30), "Event"
    Rectangle (232,12 232x35), "%s", text variable: m_Instance.in_sName
    Rectangle (574,64 62x30), "Cfg"
    Checkbox (504,20 116x30), "Local Control", variable: m_Instance.stat.bLocal
    Rectangle (505,120 30x30), "%d", text variable: m_Instance.stat.nStatus
    Button (185,400 160x30), "READ", tooltip "Single read of all commands in the configuration", input disabled if: (m_Instance.stat.bLocal = FALSE) <> 0
        OnMouseClick: execute { m_Instance.ctrl.nCommand := E_RS_COMMAND.READ; m_Instance.ctrl.bExecute := TRUE; }
    Button (350,400 160x30), "READ USER", tooltip "Single read of user command", input disabled if: (m_Instance.stat.bLocal = FALSE) <> 0
        OnMouseClick: execute { m_Instance.ctrl.nCommand := E_RS_COMMAND.READ_USER; m_Instance.ctrl.bExecute := TRUE; }
    Button (185,440 160x30), "MONITOR", tooltip "Continuously read all commands in the configuration", input disabled if: (m_Instance.stat.bLocal = FALSE) <> 0
        OnMouseClick: execute { m_Instance.ctrl.nCommand := E_RS_COMMAND.MONITOR; m_Instance.ctrl.bExecute := TRUE; }
    Button (350,440 160x30), "MONITOR USER", tooltip "Continuously read the User command", input disabled if: (m_Instance.stat.bLocal = FALSE) <> 0
        OnMouseClick: execute { m_Instance.ctrl.nCommand := E_RS_COMMAND.MONITOR_USER; m_Instance.ctrl.bExecute := TRUE; }
    Rectangle (570,153 70x25), "KRDG? C"
    Rectangle (570,178 70x25), "KRDG? D"
    Rectangle (570,203 70x25), "%s", text variable: m_Instance.cfg.cmdList_Read[3].cmd
    Rectangle (570,228 70x25), "%s", text variable: m_Instance.cfg.cmdList_Read[4].cmd
    Rectangle (570,253 70x25), "%s", text variable: m_Instance.cfg.cmdList_Read[5].cmd
    Rectangle (570,278 70x25), "%s", text variable: m_Instance.cfg.cmdList_Read[6].cmd
    Rectangle (570,303 70x25), "%s", text variable: m_Instance.cfg.cmdList_Read[7].cmd
    Rectangle (570,328 70x25), "%s", text variable: m_Instance.cfg.cmdList_Read[8].cmd
    Rectangle (570,353 70x25), "%s", text variable: m_Instance.cfg.cmdList_Read[9].cmd
    Rectangle (570,378 70x25), "%s", text variable: m_Instance.cfg.cmdList_Read[10].cmd
    Rectangle (570,403 70x25), "%s", text variable: m_Instance.cfg.cmdList_Read[11].cmd
    Rectangle (570,428 70x25), "%s", text variable: m_Instance.cfg.cmdList_Read[12].cmd
    Rectangle (570,453 70x25), "%s", text variable: m_Instance.cfg.cmdList_Read[13].cmd
    Rectangle (570,478 70x25), "%s", text variable: m_Instance.cfg.cmdList_Read[14].cmd
    Rectangle (570,503 70x25), "%s", text variable: m_Instance.cfg.cmdList_Read[15].cmd
    Rectangle (570,528 70x25), "%s", text variable: m_Instance.cfg.cmdList_Read[16].cmd
    Rectangle (650,153 70x25), "%.2f", text variable: m_Instance.stat.lrArrReadings[20].lrValue
    Rectangle (650,178 70x25), "%.2f", text variable: m_Instance.stat.lrArrReadings[21].lrValue
    Rectangle (650,203 70x25), "%.2f", text variable: m_Instance.stat.lrArrReadings[2].lrValue
    Rectangle (650,228 70x25), "%.2f", text variable: m_Instance.stat.lrArrReadings[3].lrValue
    Rectangle (720,228 70x25), "%.2f", text variable: m_Instance.stat.lrArrReadings[4].lrValue
    Rectangle (790,228 70x25), "%.2f", text variable: m_Instance.stat.lrArrReadings[5].lrValue
    Rectangle (650,253 70x25), "%.0f", text variable: m_Instance.stat.lrArrReadings[6].lrValue
    Rectangle (650,278 70x25), "%.0f", text variable: m_Instance.stat.lrArrReadings[8].lrValue
    Rectangle (650,303 70x25), "%.2f", text variable: m_Instance.stat.lrArrReadings[9].lrValue
    Rectangle (650,328 70x25), "%.2f", text variable: m_Instance.stat.lrArrReadings[10].lrValue
    Rectangle (720,353 70x25), "%.2f", text variable: m_Instance.stat.lrArrReadings[12].lrValue
    Rectangle (790,353 70x25), "%.2f", text variable: m_Instance.stat.lrArrReadings[13].lrValue
    Rectangle (650,353 70x25), "%.2f", text variable: m_Instance.stat.lrArrReadings[11].lrValue
    Rectangle (720,378 70x25), "%.2f", text variable: m_Instance.stat.lrArrReadings[15].lrValue
    Rectangle (650,403 70x25), "%.0f", text variable: m_Instance.stat.lrArrReadings[16].lrValue
    Rectangle (650,428 70x25), "%.2f", text variable: m_Instance.stat.lrArrReadings[17].lrValue
    Rectangle (650,453 70x25), "%.2f", text variable: m_Instance.stat.lrArrReadings[18].lrValue
    Rectangle (650,478 70x25), "%.2f", text variable: m_Instance.stat.lrArrReadings[19].lrValue
    Rectangle (650,503 70x25), "%.2f", text variable: m_Instance.stat.lrArrReadings[20].lrValue
    Rectangle (650,528 70x25), "%.2f", text variable: m_Instance.stat.lrArrReadings[21].lrValue
    Rectangle (654,64 62x30), "Stat"
    Button (350,300 160x30), "STOP MONITOR", tooltip "Stop Monitoring if in OP/MONITORIN state.", input disabled if: (m_Instance.stat.bLocal = FALSE) <> 0
        OnMouseClick: execute { m_Instance.ctrl.nCommand := E_RS_COMMAND.STOPMON; m_Instance.ctrl.bExecute := TRUE; }
    Rectangle (56,15 101x30), "Simulation", invisible if: (m_Instance.stat.bSimulation=FALSE)
    Ellipse (162,20 20x20), tooltip "GREEN=Initialized RED=Not-initialized", text variable: m_Instance.stat.bInitialised, invisible if: (m_Instance.stat.bSimulation=FALSE)
    Rectangle (720,253 70x25), "%.2f", text variable: m_Instance.stat.lrArrReadings[7].lrValue
    Rectangle (650,378 70x25), "%.0f", text variable: m_Instance.stat.lrArrReadings[14].lrValue
    Rectangle (570,103 70x25), "%s", text variable: m_Instance.cfg.cmdList_Read[1].cmd
    Rectangle (570,128 70x25), "%s", text variable: m_Instance.cfg.cmdList_Read[2].cmd
    Rectangle (650,103 70x25), "%.2f", text variable: m_Instance.stat.lrArrReadings[0].lrValue
    Rectangle (650,128 70x25), "%.2f", text variable: m_Instance.stat.lrArrReadings[1].lrValue
    Rectangle (720,178 178x25), "stat.lrArrReadings[21].lrValue"
    Rectangle (720,153 178x25), "stat.lrArrReadings[20].lrValue"
    Rectangle (720,128 178x25), "stat.lrArrReadings[1].lrValue"
    Rectangle (720,103 178x25), "stat.lrArrReadings[0].lrValue"
    Rectangle (290,530 101x25), "%d", text variable: m_Instance.nCommErrors
    Label (190,530 101x25), "Comm errors"
    Button (400,530 25x25), "C", input disabled if: (m_Instance.stat.bLocal = FALSE) <> 0
        OnMouseClick: execute { m_Instance.nCommErrors := 0; }
END_VISUALIZATION

// HMI/VISUs/Templates/GUI_TP_PUMPS
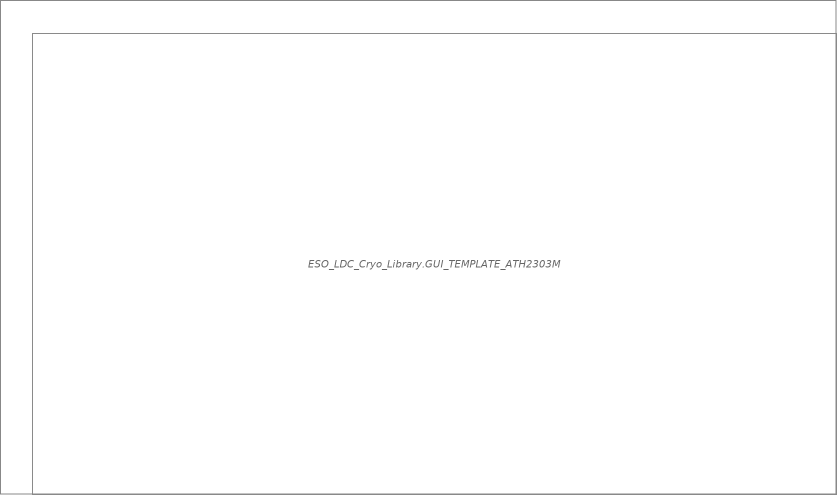
VISUALIZATION GUI_TP_PUMPS  // 837x495
    Frame (32,33 805x462)
        shows ESO_LDC_Cryo_Library.GUI_TEMPLATE_ATH2303M(m_Instance := MAIN.met_cryo_ctrl.met_evac.evac_branch_a.tp, m_bEnable := MAIN.met_cryo_ctrl.met_evac.evac_branch_a.ctrl.bEnable_TMP)
END_VISUALIZATION

// HMI/VISUs/Templates/Sim_LN2_Ctrl_inputs
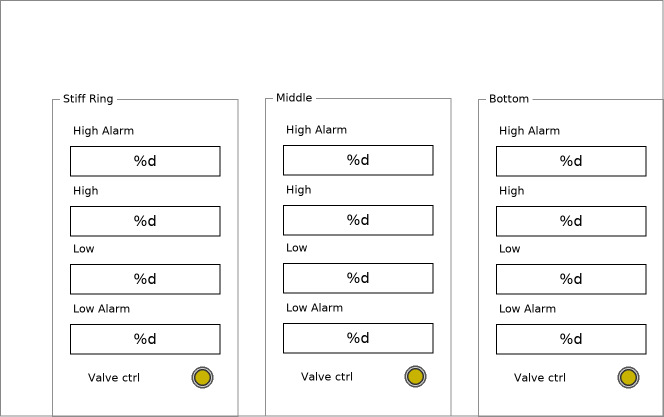
VISUALIZATION Sim_LN2_Ctrl_inputs  // 664x417
    GroupBox (52,91 186x326), "Stiff Ring"
    Rectangle (70,116 150x30), "High Alarm"
    Rectangle (70,176 150x30), "High"
    Rectangle (70,234 150x30), "Low"
    Rectangle (70,294 150x30), "Low Alarm"
    Rectangle (70,146 150x30), "%d", text variable: MAIN.met_cryo_ctrl.met_cool_down.nSim_Temp_HA_1
        OnMouseClick: write the text variable via Edit
    Rectangle (70,206 150x30), "%d", text variable: MAIN.met_cryo_ctrl.met_cool_down.nSim_Temp_H_1
        OnMouseClick: write the text variable via Edit
    Rectangle (70,264 150x30), "%d", text variable: MAIN.met_cryo_ctrl.met_cool_down.nSim_Temp_L_1
        OnMouseClick: write the text variable via Edit
    Rectangle (70,324 150x30), "%d", text variable: MAIN.met_cryo_ctrl.met_cool_down.nSim_Temp_LA_1
        OnMouseClick: write the text variable via Edit
    Lamp1 (190,365 25x25), variable: MAIN.met_cryo_ctrl.met_cool_down.lc_ln2_level_ctrl[1].LN2_Valve.Actuator.q_bCtrl, style: Lamp-Lamp1-Yellow
    Rectangle (85,363 64x30), "Valve ctrl"
    GroupBox (265,90 186x326), "Middle"
    Rectangle (283,115 150x30), "High Alarm"
    Rectangle (283,175 150x30), "High"
    Rectangle (283,233 150x30), "Low"
    Rectangle (283,293 150x30), "Low Alarm"
    Rectangle (283,145 150x30), "%d", text variable: MAIN.met_cryo_ctrl.met_cool_down.nSim_Temp_HA_2
        OnMouseClick: write the text variable via Edit
    Rectangle (283,205 150x30), "%d", text variable: MAIN.met_cryo_ctrl.met_cool_down.nSim_Temp_H_2
        OnMouseClick: write the text variable via Edit
    Rectangle (283,263 150x30), "%d", text variable: MAIN.met_cryo_ctrl.met_cool_down.nSim_Temp_L_2
        OnMouseClick: write the text variable via Edit
    Rectangle (283,323 150x30), "%d", text variable: MAIN.met_cryo_ctrl.met_cool_down.nSim_Temp_LA_2
        OnMouseClick: write the text variable via Edit
    Lamp1 (403,364 25x25), variable: MAIN.met_cryo_ctrl.met_cool_down.lc_ln2_level_ctrl[2].LN2_Valve.Actuator.q_bCtrl, style: Lamp-Lamp1-Yellow
    Rectangle (298,362 64x30), "Valve ctrl"
    GroupBox (478,91 186x326), "Bottom"
    Rectangle (496,116 150x30), "High Alarm"
    Rectangle (496,176 150x30), "High"
    Rectangle (496,234 150x30), "Low"
    Rectangle (496,294 150x30), "Low Alarm"
    Rectangle (496,146 150x30), "%d", text variable: MAIN.met_cryo_ctrl.met_cool_down.nSim_Temp_HA_3
        OnMouseClick: write the text variable via Edit
    Rectangle (496,206 150x30), "%d", text variable: MAIN.met_cryo_ctrl.met_cool_down.nSim_Temp_H_3
        OnMouseClick: write the text variable via Edit
    Rectangle (496,264 150x30), "%d", text variable: MAIN.met_cryo_ctrl.met_cool_down.nSim_Temp_L_3
        OnMouseClick: write the text variable via Edit
    Rectangle (496,324 150x30), "%d", text variable: MAIN.met_cryo_ctrl.met_cool_down.nSim_Temp_LA_3
        OnMouseClick: write the text variable via Edit
    Lamp1 (616,365 25x25), variable: MAIN.met_cryo_ctrl.met_cool_down.lc_ln2_level_ctrl[3].LN2_Valve.Actuator.q_bCtrl, style: Lamp-Lamp1-Yellow
    Rectangle (511,363 64x30), "Valve ctrl"
END_VISUALIZATION

// HMI/VISUs/Templates/TEMPLATE_AMBIENT_PRESSURE_READING
